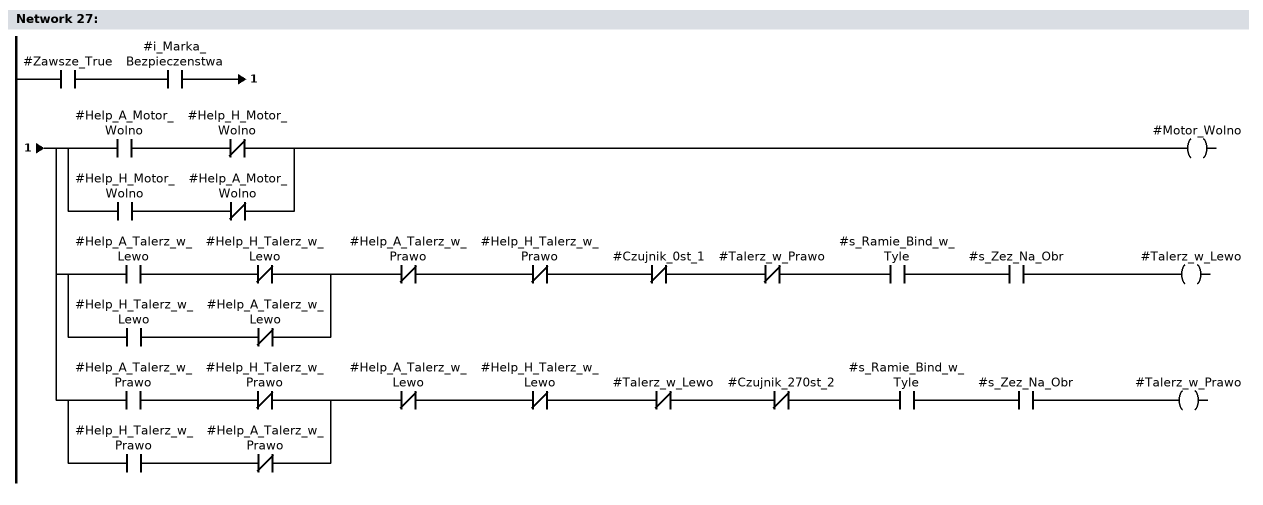
[picture p506: Obr_Na_Poz_4 networks 27-27]
NETWORK
TITLE =
//wykonianie obrotu warunki jazdy
      A     #Zawsze_True;
      A     #i_Marka_Bezpieczenstwa;
      =     L 1.0;
      A     L 1.0;
      A(;
      A     #Help_A_Motor_Wolno;
      AN    #Help_H_Motor_Wolno;
      O;
      A     #Help_H_Motor_Wolno;
      AN    #Help_A_Motor_Wolno;
      );
      =     #Motor_Wolno;
      A     L 1.0;
      A(;
      A     #Help_A_Talerz_w_Lewo;
      AN    #Help_H_Talerz_w_Lewo;
      O;
      A     #Help_H_Talerz_w_Lewo;
      AN    #Help_A_Talerz_w_Lewo;
      );
      AN    #Help_A_Talerz_w_Prawo;
      AN    #Help_H_Talerz_w_Prawo;
      AN    #Czujnik_0st_1;
      AN    #Talerz_w_Prawo;
      A     #s_Ramie_Bind_w_Tyle;
      A     #s_Zez_Na_Obr;
      =     #Talerz_w_Lewo;
      A     L 1.0;
      A(;
      A     #Help_A_Talerz_w_Prawo;
      AN    #Help_H_Talerz_w_Prawo;
      O;
      A     #Help_H_Talerz_w_Prawo;
      AN    #Help_A_Talerz_w_Prawo;
      );
      AN    #Help_A_Talerz_w_Lewo;
      AN    #Help_H_Talerz_w_Lewo;
      AN    #Talerz_w_Lewo;
      AN    #Czujnik_270st_2;
      A     #s_Ramie_Bind_w_Tyle;
      A     #s_Zez_Na_Obr;
      =     #Talerz_w_Prawo;
END_FUNCTION_BLOCK

FUNCTION_BLOCK "Pozycjonowanie_Bandy"	// FB 55
//Funcja odpowiada za jazde rolek na pozycje zgodnie z rozkazem 
VERSION : 0.1
VAR_INPUT
  i_Auto_Reczny : BOOL ;
  Stop_Bezpieczenistwa : BOOL ;
  Pozycjonuj_Lewo : BOOL ;
  Pozycjonuj_Prawo : BOOL ;
  Powrot_Poz : BOOL ;
  Foto_Przod : BOOL ;
  Foto_Tyl : BOOL ;
  i_Zez_Na_Rolki : BOOL ;
  Reset : BOOL ;
  Czas_Prawo : TIME ;
  Czas_Lewo : TIME ;
  Czas_Kontrolny : TIME ;
  Czas_Pow_Prawo : TIME ;
  Czas_Pow_Lewo : TIME ;
  Blokada_Obrotu_1 : BOOL ;
  i_Resetuj_Srodek : BOOL ;	//Przesow rolek z innego trybu
END_VAR
VAR_OUTPUT
  Potw_Pozycji : BOOL ;
  Pozycja_Lewo : BOOL ;	//Odniesienie do 0st
  Pozycja_Prawo : BOOL ;	//Odniesienie do 0st
  Pozycja_Srodek : BOOL ;
  Motor_Lewo : BOOL ;
  Motor_Prawo : BOOL ;
  Motor_Wolno : BOOL ;
  Zez_Na_Obrot : BOOL ;
  Blad_Pozycjowania : BOOL ;
END_VAR
VAR
  Pozycja_Wyjsciowa : BOOL ;
  Tim_Jazdy_Prawo : FB 20;
  Tim_Jazdy_Lewo : FB 20;
  Tim_Kon_Prawo : FB 20;	//Timmer kontrolny prawo
  Tim_Kon_Lewo : FB 20;	//Timmer kontrolny lewo
  Help_Motor_Prawo : BOOL ;
  Help_Motor_Lewo : BOOL ;
  H_Repozycj_Prawo : BOOL ;
  H_Repozycj_Lewo : BOOL ;
  Help_Motor_Wolno : BOOL ;
  H_Powr_od_Prawo_1 : BOOL ;
  H_Powr_od_Lewo_1 : BOOL ;
  H_Powr_Prawo : BOOL ;
  H_Powr_Lewo : BOOL ;
  Help_Poz_Prawo : BOOL ;
  Help_Poz_Lewo : BOOL ;
  Pozycj_Warunkowe : BOOL ;
  Skrajne_Prawo : BOOL ;
  Skrajne_Lewo : BOOL ;
  Zbocze_1 : BOOL ;
  Zbocze_2 : BOOL ;
  H6 : BOOL ;
  H7 : BOOL ;
  H8 : BOOL ;
  H9 : BOOL ;
  H10 : BOOL ;
END_VAR
VAR_TEMP
  Temp_Help_1 : BOOL ;
  Temp_Help_2 : BOOL ;
  Temp_Help_3 : BOOL ;
  Czas_Aktualny : TIME ;
END_VAR
BEGIN
NETWORK
TITLE =
      A     #Foto_Przod;
      A     #Foto_Tyl;
      A     #Pozycja_Srodek;
      A     #i_Zez_Na_Rolki;	//rolki sa odblokowane w pozycji 0st lub 180st
      =     #Pozycja_Wyjsciowa;
      O     #Help_Motor_Lewo;
      O     #Help_Motor_Prawo;
      R     #Potw_Pozycji;
//warunkowe pozycjonowanie 
NETWORK
TITLE =
//Pozycjonowanie prawo
//Pozycjonowanie w prawo
      A     #i_Zez_Na_Rolki;
      A     #Pozycjonuj_Prawo;
      A     #Pozycja_Wyjsciowa;
      S     #Help_Motor_Prawo;
      S     #Help_Motor_Wolno;
      S     #Help_Poz_Prawo;
      R     #Pozycja_Srodek;
      CALL  #Tim_Jazdy_Prawo (
           IN                       := #Help_Poz_Prawo,
           STOP                     := #Stop_Bezpieczenistwa,
           PT                       := #Czas_Prawo,
           Q_0                      := #Temp_Help_2,
           ET                       := #Czas_Aktualny);
      A     #Temp_Help_2;
      O;
      A     #Help_Poz_Prawo;
      AN    #Foto_Przod;
      S     #Pozycja_Prawo;
      S     #Potw_Pozycji;
      R     #Help_Motor_Prawo;
      R     #Help_Motor_Wolno;
      R     #Help_Poz_Prawo;
//Powrot z pozycjonowania. 
//Zjazd z fotokomorki aby zrobic ponowny najazd
      O(;
      A     #Foto_Przod;
      A     #Pozycja_Prawo;
      A     #Powrot_Poz;
      AN    #H_Powr_od_Prawo_1;
      );
      O(;
      A     #Pozycj_Warunkowe;
      );
      S     #Help_Motor_Prawo;
      S     #Help_Motor_Wolno;
      S     #H_Repozycj_Prawo;
      R     #Pozycja_Prawo;
//koniec zjazdu z fotokomorki
      AN    #Foto_Przod;
      A     #H_Repozycj_Prawo;
      R     #Help_Motor_Prawo;
      R     #Help_Motor_Wolno;
      R     #H_Repozycj_Prawo;
      S     #Skrajne_Prawo;
//powrot na pozycje na srodku obrtnicy
      A(;
      O     #Powrot_Poz;
      O     #Skrajne_Prawo;
      O     #Pozycj_Warunkowe;
      );
      A(;
      O     #Pozycja_Prawo;
      O     #Skrajne_Prawo;
      );
      AN    #Foto_Przod;
      S     #Help_Motor_Lewo;
      S     #Help_Motor_Wolno;
      S     #H_Powr_od_Prawo_1;
      R     #Help_Motor_Prawo;
      R     #Pozycja_Prawo;
      R     #Skrajne_Prawo;
      R     #Pozycj_Warunkowe;
NETWORK
TITLE =
//Pozycjonowanie lewo
//
//
//Pozycjonowanie w lewo
      A     #i_Zez_Na_Rolki;
      A     #Pozycjonuj_Lewo;
      A     #Pozycja_Wyjsciowa;
      S     #Help_Motor_Lewo;
      S     #Help_Motor_Wolno;
      S     #Help_Poz_Lewo;
      R     #Pozycja_Srodek;
      CALL  #Tim_Jazdy_Lewo (
           IN                       := #Help_Poz_Lewo,
           STOP                     := #Stop_Bezpieczenistwa,
           PT                       := #Czas_Lewo,
           Q_0                      := #Temp_Help_2,
           ET                       := #Czas_Aktualny);
      A     #Temp_Help_2;
      O;
      AN    #Foto_Tyl;
      A     #Help_Poz_Lewo;
      S     #Pozycja_Lewo;
      S     #Potw_Pozycji;
      R     #Help_Motor_Lewo;
      R     #Help_Motor_Wolno;
      R     #Help_Poz_Lewo;
//Powrot z pozycjonowania. 
//Zjazd z fotokomorki aby zrobic ponowny najazd
      A     #Foto_Tyl;
      A     #Pozycja_Lewo;
      A     #Powrot_Poz;
      AN    #H_Powr_od_Lewo_1;
      S     #Help_Motor_Lewo;
      S     #Help_Motor_Wolno;
      S     #H_Repozycj_Lewo;
      R     #Potw_Pozycji;
//koniec zjazdu z fotokomorki
      AN    #Foto_Tyl;
      A     #H_Repozycj_Lewo;
      R     #Help_Motor_Lewo;
      R     #Help_Motor_Wolno;
      R     #H_Repozycj_Lewo;
      S     #Skrajne_Lewo;
//powrot na pozycje na srodku obrotnicy
      O     #Skrajne_Lewo;
      O(;
      A     #Powrot_Poz;
      A     #Pozycja_Lewo;
      );
      AN    #Foto_Tyl;
      S     #Help_Motor_Prawo;
      S     #Help_Motor_Wolno;
      S     #H_Powr_od_Lewo_1;
      R     #Help_Motor_Lewo;
      R     #Pozycja_Lewo;
      R     #Skrajne_Lewo;
NETWORK
TITLE =
//Okreselnie srodka
//Jazda  powrotna w strone prawa do œrodka
      A     #Foto_Przod;
      A     #H_Powr_od_Prawo_1;
      S     #H_Powr_Prawo;
      CALL  #Tim_Kon_Prawo (
           IN                       := #H_Powr_Prawo,
           STOP                     := #Stop_Bezpieczenistwa,
           PT                       := #Czas_Pow_Prawo,
           Q_0                      := #Temp_Help_2,
           ET                       := #Czas_Aktualny);
      A     #Foto_Tyl;
      A     #H_Powr_od_Lewo_1;
      S     #H_Powr_Lewo;
      CALL  #Tim_Kon_Lewo (
           IN                       := #H_Powr_Lewo,
           STOP                     := #Stop_Bezpieczenistwa,
           PT                       := #Czas_Pow_Lewo,
           Q_0                      := #Temp_Help_3,
           ET                       := #Czas_Aktualny);
//nieautoryzowane kasowanie srodka
      A     #i_Resetuj_Srodek;
      FP    #Zbocze_2;
      R     #Pozycja_Srodek;
      O     #Temp_Help_3;
      O     #Temp_Help_2;
      S     #Pozycja_Srodek;
      S     #Potw_Pozycji;
      R     #Pozycj_Warunkowe;
//zresetuj bity i pozycjonuj do srodka
      A     #Reset;
      FP    #Zbocze_1;
      S     #Pozycj_Warunkowe;
      R     #Pozycja_Srodek;
      R     #Potw_Pozycji;
      =     #Temp_Help_1;
      O     #Temp_Help_1;
      O     #Temp_Help_2;
      O     #Temp_Help_3;
      R     #Help_Motor_Prawo;
      R     #Help_Motor_Lewo;
      R     #Help_Motor_Wolno;
      R     #H_Powr_od_Prawo_1;
      R     #H_Powr_od_Lewo_1;
      R     #H_Repozycj_Prawo;
      R     #H_Repozycj_Lewo;
      R     #Help_Poz_Prawo;
      R     #Help_Poz_Lewo;
      R     #Skrajne_Prawo;
      R     #Skrajne_Lewo;
      R     #H_Powr_Prawo;
      R     #H_Powr_Lewo;
      R     #Pozycja_Prawo;
      R     #Pozycja_Lewo;
NETWORK
TITLE =
//Przyporzadkowanie wyjsc
      A     #i_Auto_Reczny;
      A     #i_Zez_Na_Rolki;
      A     #Help_Motor_Lewo;
      =     #Motor_Lewo;
      A     #i_Auto_Reczny;
      A     #i_Zez_Na_Rolki;
      A     #Help_Motor_Prawo;
      =     #Motor_Prawo;
      A     #i_Auto_Reczny;
      A     #Help_Motor_Wolno;
      =     #Motor_Wolno;
//Zezwolenie na obrot obrotnicy
      A(;
      A     #Foto_Przod;
      A     #Foto_Tyl;
      O;
      AN    #Foto_Przod;
      AN    #Foto_Tyl;
      );
      A     #Blokada_Obrotu_1;
      =     #Zez_Na_Obrot;
END_FUNCTION_BLOCK

FUNCTION_BLOCK "Bindownica_Test"	// FB 57
VERSION : 0.1
VAR_INPUT
  i_Bind_Obwod_Ok : BOOL ;	//270 stopni
  i_Bind_Poz_Podst : BOOL ;
  i_Bind_Syg_Got : BOOL ;
  i_Bind_Blad : BOOL ;
  i_Bind_Start_Kon : BOOL ;	//Bindownica start koniec wiazania
  i_Przesznuruj : BOOL ;	//Przesznurowanie imituje bindownice
  i_Cykl_Bindowanie : BOOL ;
END_VAR
VAR_OUTPUT
  io_Bind_Obwod_Ok : BOOL ;	//270 stopni
  io_Bind_Poz_Podst : BOOL ;
  io_Bind_Syg_Got : BOOL ;
  io_Bind_Blad : BOOL ;
  io_Bind_Start_Kon : BOOL ;	//Bindownica start koniec wiazania
END_VAR
VAR
  CZas_Testowy : SFB 4;
END_VAR
VAR_TEMP
  temp_help_1 : BOOL ;
END_VAR
BEGIN
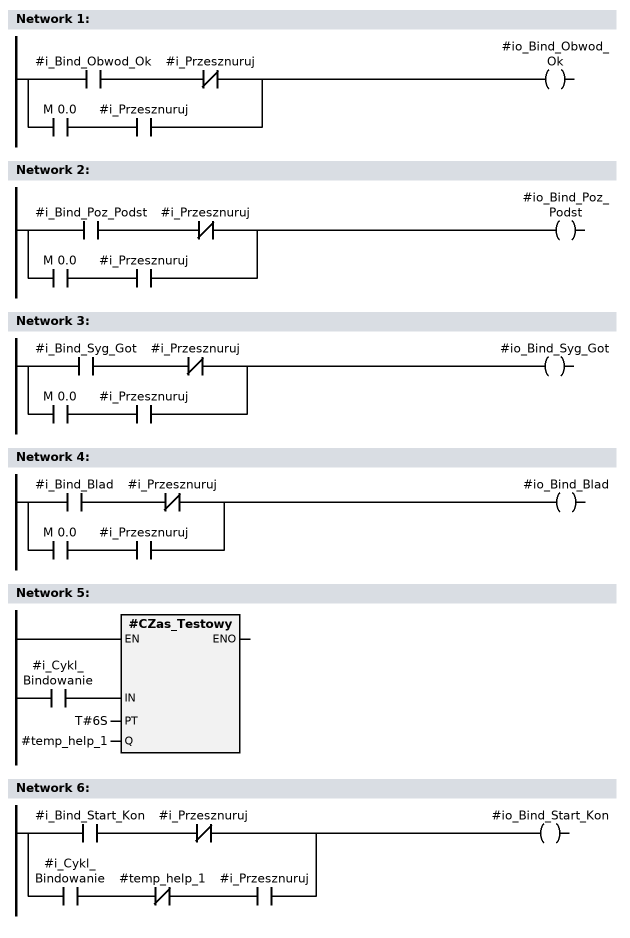
NETWORK
TITLE =
//bind obwod ok
      A     #i_Bind_Obwod_Ok;
      AN    #i_Przesznuruj;
      O;
      A     M 0.0;
      A     #i_Przesznuruj;
      =     #io_Bind_Obwod_Ok;
NETWORK
TITLE =
//Pozycja podstawowa
      A     #i_Bind_Poz_Podst;
      AN    #i_Przesznuruj;
      O;
      A     M 0.0;
      A     #i_Przesznuruj;
      =     #io_Bind_Poz_Podst;
NETWORK
TITLE =
//sygnal gotowosc
      A     #i_Bind_Syg_Got;
      AN    #i_Przesznuruj;
      O;
      A     M 0.0;
      A     #i_Przesznuruj;
      =     #io_Bind_Syg_Got;
NETWORK
TITLE =
//Blad bindowania
      A     #i_Bind_Blad;
      AN    #i_Przesznuruj;
      O;
      A     M 0.0;
      A     #i_Przesznuruj;
      =     #io_Bind_Blad;
NETWORK
TITLE =
//bindowanie
//
      A     #i_Cykl_Bindowanie;
      =     L 1.0;
      BLD   103;
      CALL  #CZas_Testowy (
           IN                       := L 1.0,
           PT                       := T#6S,
           Q                        := #temp_help_1);
      NOP   0;
NETWORK
TITLE =
//start koniec bindowania
      A     #i_Bind_Start_Kon;
      AN    #i_Przesznuruj;
      O;
      A     #i_Cykl_Bindowanie;
      AN    #temp_help_1;
      A     #i_Przesznuruj;
      =     #io_Bind_Start_Kon;
END_FUNCTION_BLOCK

FUNCTION_BLOCK "Pozycjonowanie_Palety"	// FB 58
//Funcja odpowiada za jazde rolek na pozycje zgodnie z rozkazem. Zmiany do wersji 
//porzednie:
//
//-o powrocie z pozycjonowania gdy stan pozycji palety jest nieustalony decyduje
// bit wejsciowy reset
//
VERSION : 0.1
VAR_INPUT
  i_Marka_Bezpieczenstwa : BOOL ;
  i_Rezerwa : BOOL ;
  i_Auto_Reczny : BOOL ;
  i_Pozycjonuj_Lewo : BOOL ;
  i_Pozycjonuj_Prawo : BOOL ;
  i_Pozycjonuj_Srodek : BOOL ;
  i_Foto_Przod : BOOL ;
  i_Foto_Tyl : BOOL ;
  s_i_Zez_Na_Rolki : BOOL ;
  i_Czas_Jazdy_Prawo : TIME ;
  i_Czas_Jazdy_Lewo : TIME ;
  i_Czas_Opoznienia : TIME ;
  i_Czas_Powrotu_Prawo : TIME ;
  i_Czas_Powrotu_Lewo : TIME ;
  s_i_Blokada_Obrotu : BOOL ;
  i_Resetuj_Srodek : BOOL ;	//Resetowanie zewnetrzne konca palety
  i_Setuj_Srodek : BOOL ;	//Ustawienie zewnetrzne srodka palety
END_VAR
VAR_OUTPUT
  o_Pozycja_Lewo : BOOL ;	//Odniesienie do 0st
  o_Pozycja_Prawo : BOOL ;	//Odniesienie do 0st
  o_Pozycja_Srodek : BOOL ;
  o_Potw_Pozycji : BOOL ;
  o_Motor_Lewo : BOOL ;
  o_Motor_Prawo : BOOL ;
  o_Motor_Wolno : BOOL ;
  s_o_Zez_Na_Obrot : BOOL ;
  o_Rezerwa_1 : BOOL ;
  o_Rezerwa_2 : BOOL ;
  o_Rezerwa_3 : BOOL ;
END_VAR
VAR
  Tim_Jazdy_Lewo : FB 20;
  Tim_Jazdy_Prawo : FB 20;
  Tim_Kon_Prawo : FB 20;	//Timmer kontrolny prawo
  Tim_Kon_Lewo : FB 20;	//Timmer kontrolny lewo
  Tim_Opoznienia : FB 20;
  Stop_Czas_Kontrolny : BOOL ;
  Help_Motor_Prawo : BOOL ;
  Help_Motor_Lewo : BOOL ;
  Help_Motor_Wolno : BOOL ;
  H_Repozycj_Prawo : BOOL ;
  H_Repozycj_Lewo : BOOL ;
  H_Powrot_od_Prawej : BOOL ;
  H_Powrot_od_Lewej : BOOL ;
  H_Czas_Powr_Prawo : BOOL ;
  H_Czas_Powr_Lewo : BOOL ;
  H_Czas_Jazdy_Prawo : BOOL ;
  H_Czas_Jazdy_Lewo : BOOL ;
  H_Krawedz_Prawo : BOOL ;
  H_Krawedz_Lewo : BOOL ;
  H_Pozycja_Wyjsciowa : BOOL ;
  H_Brak_Pozycji : BOOL ;
  Zbocze_1 : BOOL ;
  Zbocze_2 : BOOL ;
  H_Jakas_Pozycja : BOOL ;
  H8 : BOOL ;
  H9 : BOOL ;
  H10 : BOOL ;
  H11 : BOOL ;
  H12 : BOOL ;
END_VAR
VAR_TEMP
  Temp_Help_1 : BOOL ;
  Temp_Help_2 : BOOL ;
  Temp_Help_3 : BOOL ;
  Temp_Help_4 : BOOL ;
  Czas_Aktualny : TIME ;
END_VAR
BEGIN
NETWORK
TITLE =
//Ten network celowo ma byc wolny
NETWORK
TITLE =
//Zatrzymanie czasu w timmerach gdy obwod bezpieczenstwa nie ok
      A     #i_Marka_Bezpieczenstwa;
      S     #Stop_Czas_Kontrolny;
      AN    #i_Marka_Bezpieczenstwa;
      AN    #Stop_Czas_Kontrolny;
      JC    end;
      AN    #i_Marka_Bezpieczenstwa;
      R     #Stop_Czas_Kontrolny;
NETWORK
TITLE =
      A     #i_Foto_Przod;
      A     #i_Foto_Tyl;
      A     #o_Pozycja_Srodek;
      A     #s_i_Zez_Na_Rolki;	//rolki sa odblokowane w pozycji 0st lub 180st
      =     #H_Pozycja_Wyjsciowa;
//Reset pozycji gdy silnki wykonaja ruch
      O     #Help_Motor_Lewo;
      O     #Help_Motor_Prawo;
      R     #o_Pozycja_Prawo;
      R     #o_Pozycja_Srodek;
      R     #o_Pozycja_Lewo;
//warunkowe pozycjonowanie brak pozycji
      AN    #o_Pozycja_Prawo;
      AN    #o_Pozycja_Lewo;
      AN    #o_Pozycja_Srodek;
      =     #H_Brak_Pozycji;
      NOT;
      =     #H_Jakas_Pozycja;
NETWORK
TITLE =
//Pozycjonowanie prawo
//Pozycjonowanie w prawo
      A     #i_Pozycjonuj_Prawo;
      AN    #i_Pozycjonuj_Srodek;
      AN    #i_Pozycjonuj_Lewo;
      A     #H_Pozycja_Wyjsciowa;
      S     #Help_Motor_Prawo;
      R     #Help_Motor_Lewo;
      S     #H_Czas_Jazdy_Prawo;
//Uruchom zjazd z fotokomorki
      CALL  #Tim_Jazdy_Prawo (
           IN                       := #H_Czas_Jazdy_Prawo,
           STOP                     := #Stop_Czas_Kontrolny,
           PT                       := #i_Czas_Jazdy_Prawo,
           Q_0                      := #Temp_Help_2,
           ET                       := #Czas_Aktualny);
      A     #Temp_Help_2;
      O;
      A     #H_Czas_Jazdy_Prawo;
      AN    #i_Foto_Przod;
      S     #o_Pozycja_Prawo;
      R     #Help_Motor_Prawo;
      R     #H_Czas_Jazdy_Prawo;
NETWORK
TITLE =
//Powrot ze strony prawej
//Powrot z pozycjonowania. 
//Zjazd z fotokomorki aby zrobic ponowny najazd
      O     #o_Pozycja_Prawo;
      O     #H_Brak_Pozycji;
      A     #i_Pozycjonuj_Srodek;
      A     #i_Foto_Przod;
      A     #i_Foto_Tyl;
      A     #s_i_Zez_Na_Rolki;
      AN    #H_Powrot_od_Prawej;
      S     #Help_Motor_Prawo;
      S     #H_Repozycj_Prawo;
      R     #Help_Motor_Lewo;
//koniec zjazdu z fotokomorki
      AN    #i_Foto_Przod;
//      A     #H_Repozycj_Prawo
      R     #Help_Motor_Prawo;
      R     #H_Repozycj_Prawo;
      S     #H_Krawedz_Prawo;
//powrot na pozycje na srodku obrotnicy
      A(;
      O     #i_Pozycjonuj_Srodek;
      O     #H_Krawedz_Prawo;
      );
      A(;
      O     #o_Pozycja_Prawo;
      O     #H_Krawedz_Prawo;
      );
      AN    #i_Foto_Przod;
      S     #Help_Motor_Lewo;
      S     #H_Powrot_od_Prawej;
      R     #Help_Motor_Prawo;
      R     #H_Krawedz_Prawo;
NETWORK
TITLE =
//Pozycjonowanie lewo
//
//
//Pozycjonowanie w lewo
      A     #i_Pozycjonuj_Lewo;
      AN    #i_Pozycjonuj_Srodek;
      AN    #i_Pozycjonuj_Prawo;
      A     #H_Pozycja_Wyjsciowa;
      S     #Help_Motor_Lewo;
      R     #Help_Motor_Prawo;
      S     #H_Czas_Jazdy_Lewo;
      CALL  #Tim_Jazdy_Lewo (
           IN                       := #H_Czas_Jazdy_Lewo,
           STOP                     := #Stop_Czas_Kontrolny,
           PT                       := #i_Czas_Jazdy_Lewo,
           Q_0                      := #Temp_Help_2,
           ET                       := #Czas_Aktualny);
      A     #Temp_Help_2;
      O;
      A     #H_Czas_Jazdy_Lewo;
      AN    #i_Foto_Tyl;
      S     #o_Pozycja_Lewo;
      R     #Help_Motor_Lewo;
      R     #H_Czas_Jazdy_Lewo;
NETWORK
TITLE =
//Powrot ze strony lewej
//Powrot z pozycjonowania. 
//Zjazd z fotokomorki aby zrobic ponowny najazd
      A     #i_Pozycjonuj_Srodek;
      A     #i_Foto_Przod;
      A     #i_Foto_Tyl;
      A     #o_Pozycja_Lewo;
      A     #s_i_Zez_Na_Rolki;
      AN    #H_Powrot_od_Lewej;
      S     #Help_Motor_Lewo;
      R     #Help_Motor_Prawo;
      S     #H_Repozycj_Lewo;
//koniec zjazdu z fotokomorki
      AN    #i_Foto_Tyl;
      A     #H_Repozycj_Lewo;
      R     #Help_Motor_Lewo;
      R     #H_Repozycj_Lewo;
      S     #H_Krawedz_Lewo;
//powrot na pozycje na srodku obrotnicy
      O     #H_Krawedz_Lewo;
      O(;
      A     #i_Pozycjonuj_Srodek;
      A     #o_Pozycja_Lewo;
      );
      AN    #i_Foto_Tyl;
      S     #Help_Motor_Prawo;
      S     #H_Powrot_od_Lewej;
      R     #Help_Motor_Lewo;
      R     #H_Krawedz_Lewo;
NETWORK
TITLE =
//Okreselnie srodka
//Jazda  powrotna w strone prawa do œrodka
      A     #i_Foto_Przod;
      A     #H_Powrot_od_Prawej;
      S     #H_Czas_Powr_Prawo;
      CALL  #Tim_Kon_Prawo (
           IN                       := #H_Czas_Powr_Prawo,
           STOP                     := #Stop_Czas_Kontrolny,
           PT                       := #i_Czas_Powrotu_Prawo,
           Q_0                      := #Temp_Help_1,
           ET                       := #Czas_Aktualny);
//Powrot ze strony lewej do srodka
      A     #i_Foto_Tyl;
      A     #H_Powrot_od_Lewej;
      S     #H_Czas_Powr_Lewo;
      CALL  #Tim_Kon_Lewo (
           IN                       := #H_Czas_Powr_Lewo,
           STOP                     := #Stop_Czas_Kontrolny,
           PT                       := #i_Czas_Powrotu_Lewo,
           Q_0                      := #Temp_Help_2,
           ET                       := #Czas_Aktualny);
//nieautoryzowane kasowanie srodka
      A     #i_Resetuj_Srodek;
      R     #o_Pozycja_Srodek;
      =     #Temp_Help_3;
//nieautoryzowane setowanie  srodka
      A     #i_Setuj_Srodek;
      FP    #Zbocze_1;
      A     #i_Foto_Przod;
      A     #i_Foto_Tyl;
      S     #o_Pozycja_Srodek;
      =     #Temp_Help_4;
      O     #Temp_Help_1;
      O     #Temp_Help_2;
      S     #o_Pozycja_Srodek;
//Reset wszystkich zbedncyh bitow
      O     #Temp_Help_1;
      O     #Temp_Help_2;
      O     #Temp_Help_3;
      O     #Temp_Help_4;
      R     #Help_Motor_Prawo;
      R     #Help_Motor_Lewo;
      R     #H_Powrot_od_Prawej;
      R     #H_Powrot_od_Lewej;
      R     #H_Repozycj_Prawo;
      R     #H_Repozycj_Lewo;
      R     #H_Czas_Jazdy_Prawo;
      R     #H_Czas_Jazdy_Lewo;
      R     #H_Krawedz_Prawo;
      R     #H_Krawedz_Lewo;
      R     #H_Czas_Powr_Prawo;
      R     #H_Czas_Powr_Lewo;
      R     #o_Pozycja_Prawo;
      R     #o_Pozycja_Lewo;
NETWORK
TITLE =
//Jezeli dluzej niz 1.5 sekundy to pozycja potwierdzona
      CALL  #Tim_Opoznienia (
           IN                       := #H_Jakas_Pozycja,
           STOP                     := #Stop_Czas_Kontrolny,
           PT                       := T#1S500MS,
           Q_0                      := #o_Potw_Pozycji);
NETWORK
TITLE =
//Przyporzadkowanie wyjsc
end:  NOP   0;
//-
      A     #i_Auto_Reczny;
      A     #i_Marka_Bezpieczenstwa;
      A     #s_i_Zez_Na_Rolki;
      A     #Help_Motor_Lewo;
      AN    #Help_Motor_Prawo;
      =     #o_Motor_Lewo;
//-
      A     #i_Auto_Reczny;
      A     #i_Marka_Bezpieczenstwa;
      A     #s_i_Zez_Na_Rolki;
      A     #Help_Motor_Prawo;
      AN    #Help_Motor_Lewo;
      =     #o_Motor_Prawo;
//-
      O     #o_Motor_Lewo;
      O     #o_Motor_Prawo;
      =     #o_Motor_Wolno;
//Zezwolenie na obrot obrotnicy
      A(;
      A     #i_Foto_Przod;
      A     #i_Foto_Tyl;
      O;
      AN    #i_Foto_Przod;
      AN    #i_Foto_Tyl;
      );
      A     #s_i_Blokada_Obrotu;
      =     #s_o_Zez_Na_Obrot;
END_FUNCTION_BLOCK

FUNCTION "Funkcja_Bezpieczenstwa" : VOID	// FC 3
//Funkcja steruje bezpieczenstwem maszyny
VERSION : 0.1
VAR_TEMP
  Help_Bit : BOOL ;
END_VAR
BEGIN
NETWORK
TITLE =
//Ten Network celowo jest wolny
//
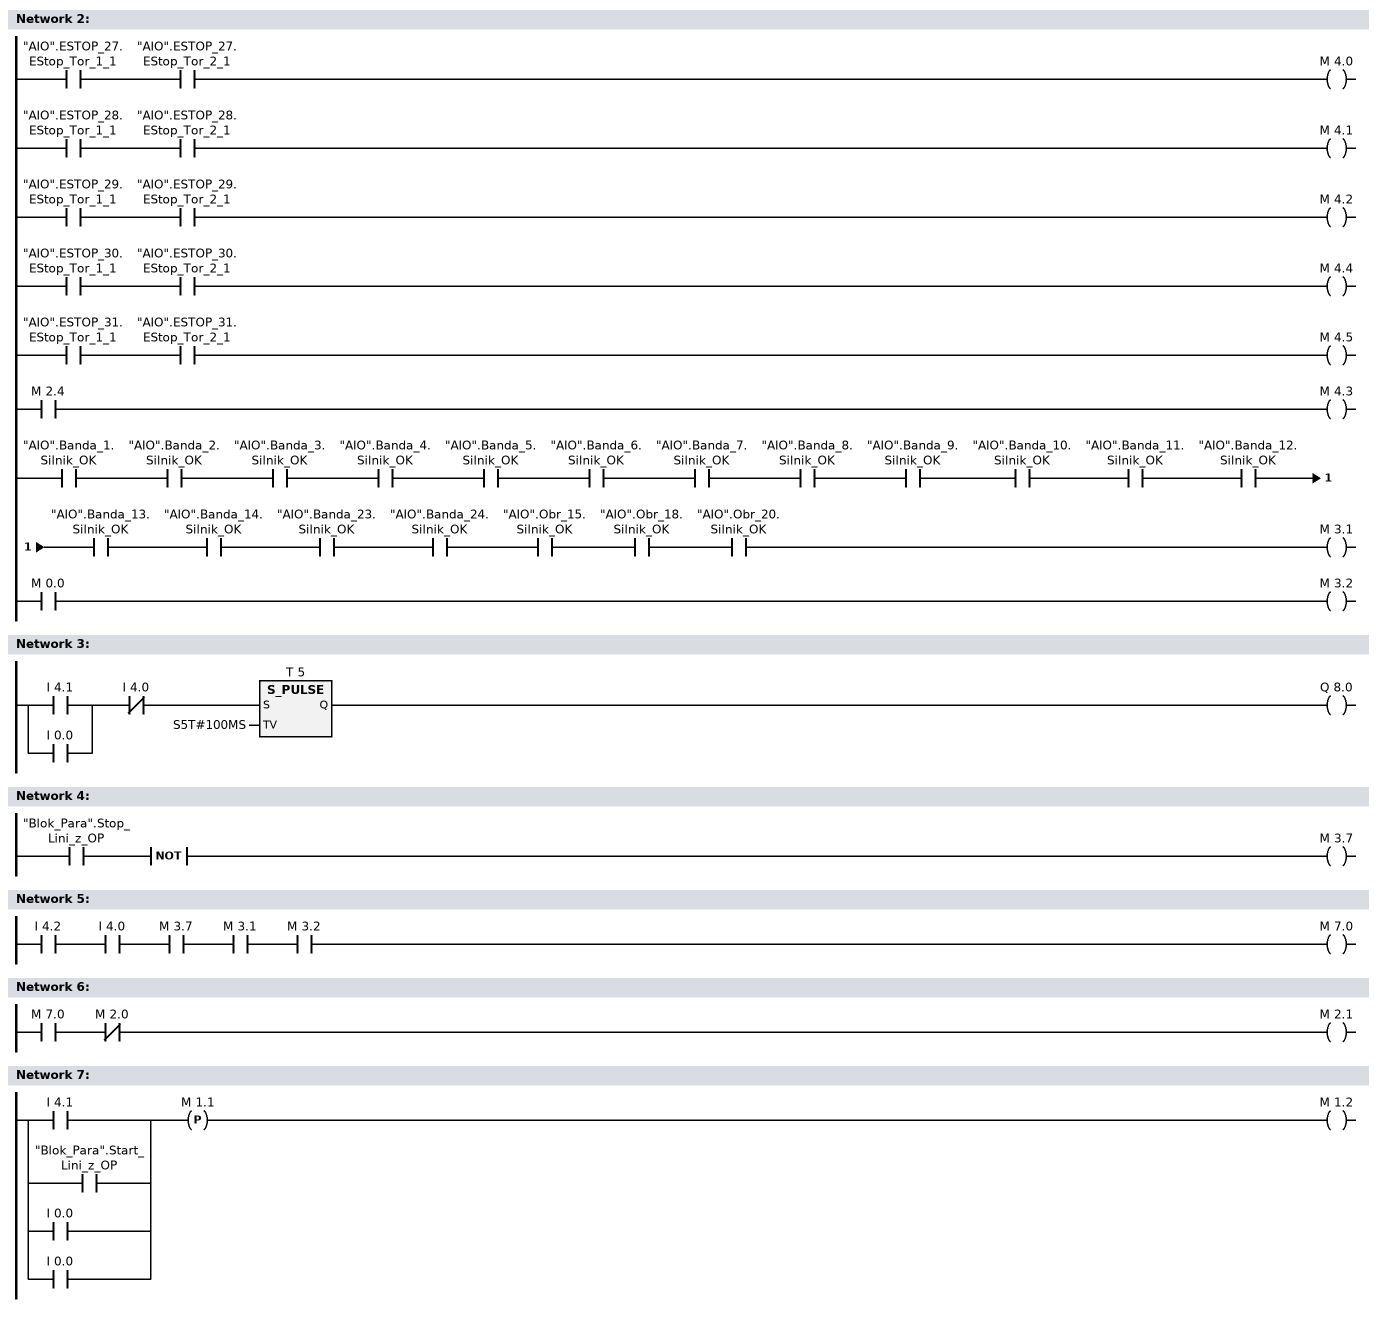
NETWORK
TITLE =
//Not Aus 27*******************************
      A     "AIO".ESTOP_27.EStop_Tor_1_1;
      A     "AIO".ESTOP_27.EStop_Tor_2_1;
      =     M 4.0;
//Not Aus 28*******************************
      A     "AIO".ESTOP_28.EStop_Tor_1_1;
      A     "AIO".ESTOP_28.EStop_Tor_2_1;
      =     M 4.1;
//Not Aus 29*******************************
      A     "AIO".ESTOP_29.EStop_Tor_1_1;
      A     "AIO".ESTOP_29.EStop_Tor_2_1;
      =     M 4.2;
//Not Aus 30*******************************
      A     "AIO".ESTOP_30.EStop_Tor_1_1;
      A     "AIO".ESTOP_30.EStop_Tor_2_1;
      =     M 4.4;
//Not Aus 31*******************************
      A     "AIO".ESTOP_31.EStop_Tor_1_1;
      A     "AIO".ESTOP_31.EStop_Tor_2_1;
      =     M 4.5;
//Strefa *******************************
      A     M 2.4;
      =     M 4.3;
//Falowniki********************************
      A     "AIO".Banda_1.Silnik_OK;
      A     "AIO".Banda_2.Silnik_OK;
      A     "AIO".Banda_3.Silnik_OK;
      A     "AIO".Banda_4.Silnik_OK;
      A     "AIO".Banda_5.Silnik_OK;
      A     "AIO".Banda_6.Silnik_OK;
      A     "AIO".Banda_7.Silnik_OK;
      A     "AIO".Banda_8.Silnik_OK;
      A     "AIO".Banda_9.Silnik_OK;
      A     "AIO".Banda_10.Silnik_OK;
      A     "AIO".Banda_11.Silnik_OK;
      A     "AIO".Banda_12.Silnik_OK;
      A     "AIO".Banda_13.Silnik_OK;
      A     "AIO".Banda_14.Silnik_OK;
      A     "AIO".Banda_23.Silnik_OK;
      A     "AIO".Banda_24.Silnik_OK;
      A     "AIO".Obr_15.Silnik_OK;
      A     "AIO".Obr_18.Silnik_OK;
      A     "AIO".Obr_20.Silnik_OK;
      =     M 3.1;
//Bezpieczniki Szafa************************
//Brak w szafie bepiecznikow z kontrola wiec
      A     M 0.0;
      =     M 3.2;
NETWORK
TITLE =
//Reset przekaznika bezp
      A(;
      O     I 4.1;
      O     I 0.0;
      );
      AN    I 4.0;
      L     S5T#100MS;
      SP    T 5;
      NOP   0;
      NOP   0;
      NOP   0;
      A     T 5;
      =     Q 8.0;
NETWORK
TITLE =
      A     "Blok_Para".Stop_Lini_z_OP;
      NOT;
      =     M 3.7;
NETWORK
TITLE =
//Warunki Startu 
      A     I 4.2;
      A     I 4.0;
      A     M 3.7;
      A     M 3.1;
      A     M 3.2;
      =     M 7.0;
NETWORK
TITLE =
//warunki do strartu ok ale start nie wcisniety
      A     M 7.0;
      AN    M 2.0;
      =     M 2.1;
NETWORK
TITLE =
//Start na szafie glownej
      A(;
      O     I 4.1;
      O     "Blok_Para".Start_Lini_z_OP;
      O     I 0.0;
      O     I 0.0;
      );
      FP    M 1.1;
      =     M 1.2;
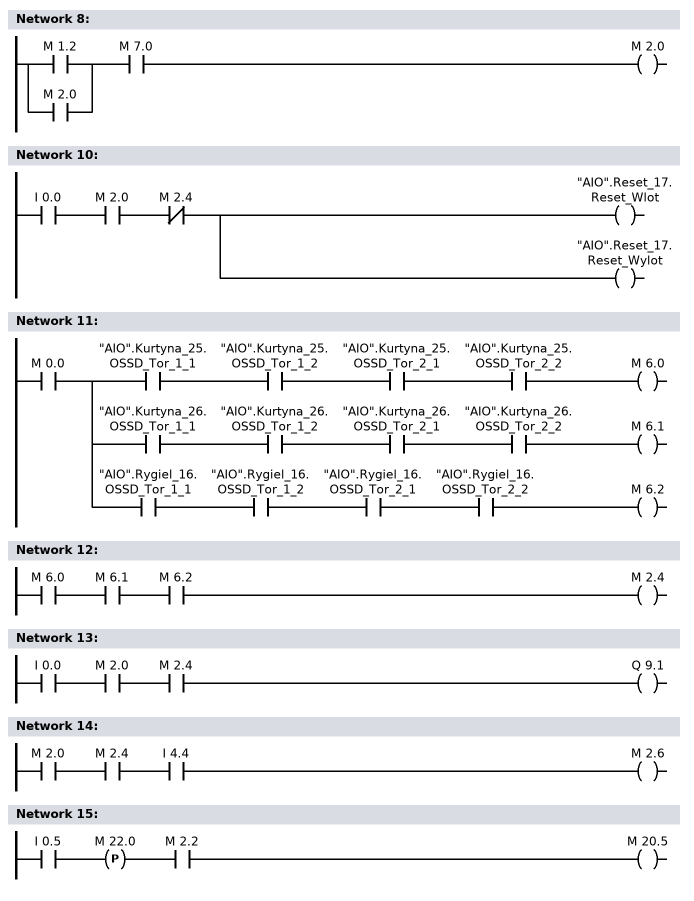
NETWORK
TITLE =
//Start Lini. Zalaczenie marki bezpieczenstwa
      A(;
      O     M 1.2;
      O     M 2.0;
      );
      A     M 7.0;
      =     M 2.0;
NETWORK
TITLE =
//Poczatek drugiego przekaznika bezpieczenstwa
NETWORK
TITLE =
//Resetowanie kurtyn bezpieczenstwa
//
      A     I 0.0;
      A     M 2.0;
      AN    M 2.4;
      =     "AIO".Reset_17.Reset_Wlot;
      =     "AIO".Reset_17.Reset_Wylot;
NETWORK
TITLE =
//Kurtyny wlot ok modul 25
//Kurtyny wylot ok modull 26
//Rygiel adres 16 ok
      A     M 0.0;
      =     L 1.0;
      A     L 1.0;
      A     "AIO".Kurtyna_25.OSSD_Tor_1_1;
      A     "AIO".Kurtyna_25.OSSD_Tor_1_2;
      A     "AIO".Kurtyna_25.OSSD_Tor_2_1;
      A     "AIO".Kurtyna_25.OSSD_Tor_2_2;
      =     M 6.0;
      A     L 1.0;
      A     "AIO".Kurtyna_26.OSSD_Tor_1_1;
      A     "AIO".Kurtyna_26.OSSD_Tor_1_2;
      A     "AIO".Kurtyna_26.OSSD_Tor_2_1;
      A     "AIO".Kurtyna_26.OSSD_Tor_2_2;
      =     M 6.1;
      A     L 1.0;
      A     "AIO".Rygiel_16.OSSD_Tor_1_1;
      A     "AIO".Rygiel_16.OSSD_Tor_1_2;
      A     "AIO".Rygiel_16.OSSD_Tor_2_1;
      A     "AIO".Rygiel_16.OSSD_Tor_2_2;
      =     M 6.2;
NETWORK
TITLE =
//Sprawdzenei czy strefa maszyny bindujacej bezpieczna
      A     M 6.0;
      A     M 6.1;
      A     M 6.2;
      =     M 2.4;
NETWORK
TITLE =
//Reset strefy bezpieczenstwa
      A     I 0.0;
      A     M 2.0;
      A     M 2.4;
      =     Q 9.1;
NETWORK
TITLE =
//Marka do pracy dla lini bindujacej
//Uwzglednione sa warunki kurtyn
//
      A     M 2.0;
      A     M 2.4;
      A     I 4.4;
      =     M 2.6;
NETWORK
TITLE =
//Tak aby potwierdzic stop gdy paleta na obrotnicy
      A     I 0.5;
      FP    M 22.0;
      A     M 2.2;
      =     M 20.5;
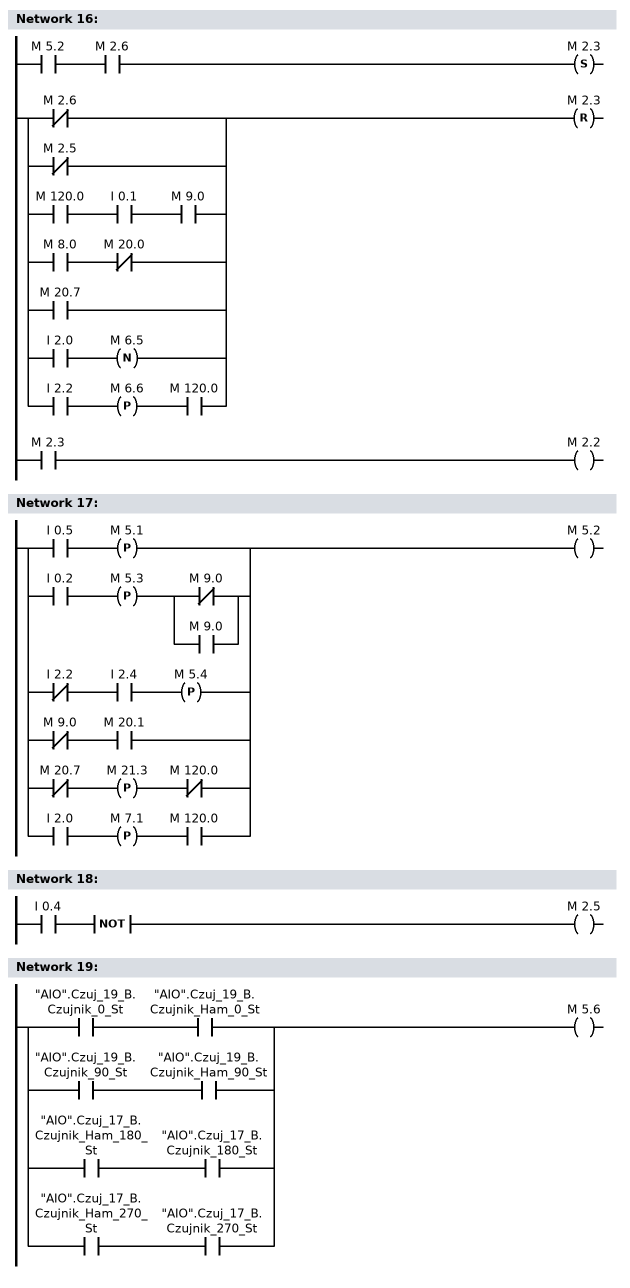
NETWORK
TITLE =
      A     M 5.2;
      A     M 2.6;
      S     M 2.3;
      A(;
      ON    M 2.6;
      ON    M 2.5;
      O(;
      A     M 120.0;
      A     I 0.1;
      A     M 9.0;
      );
      O(;
      A     M 8.0;
      AN    M 20.0;
      );
      O     M 20.7;
      O(;
      A     I 2.0;
      FN    M 6.5;
      );
      O(;
      A     I 2.2;
      FP    M 6.6;
      A     M 120.0;
      );
      );
      R     M 2.3;
      A     M 2.3;
      =     M 2.2;
NETWORK
TITLE =
//Cykl bindownicy przywrocenie
//Jest wiele drog do tego samego celu 
      A     I 0.5;
      FP    M 5.1;
      O(;
      A     I 0.2;
      FP    M 5.3;
      A(;
      ON    M 9.0;
      O     M 9.0;
      );
      );
      O(;
      AN    I 2.2;
      A     I 2.4;
      FP    M 5.4;
      );
      O(;
      AN    M 9.0;
      A     M 20.1;
      );
      O(;
      AN    M 20.7;
      FP    M 21.3;
      AN    M 120.0;
      );
      O(;
      A     I 2.0;
      FP    M 7.1;
      A     M 120.0;
      );
      =     M 5.2;
NETWORK
TITLE =
//Przycisk stop w automacie zatrzymuje maszyne 
      A     I 0.4;
      NOT;
      =     M 2.5;
NETWORK
TITLE =
//Wysuniecie OK
      A     "AIO".Czuj_19_B.Czujnik_0_St;
      A     "AIO".Czuj_19_B.Czujnik_Ham_0_St;
      O;
      A     "AIO".Czuj_19_B.Czujnik_90_St;
      A     "AIO".Czuj_19_B.Czujnik_Ham_90_St;
      O;
      A     "AIO".Czuj_17_B.Czujnik_Ham_180_St;
      A     "AIO".Czuj_17_B.Czujnik_180_St;
      O;
      A     "AIO".Czuj_17_B.Czujnik_Ham_270_St;
      A     "AIO".Czuj_17_B.Czujnik_270_St;
      =     M 5.6;
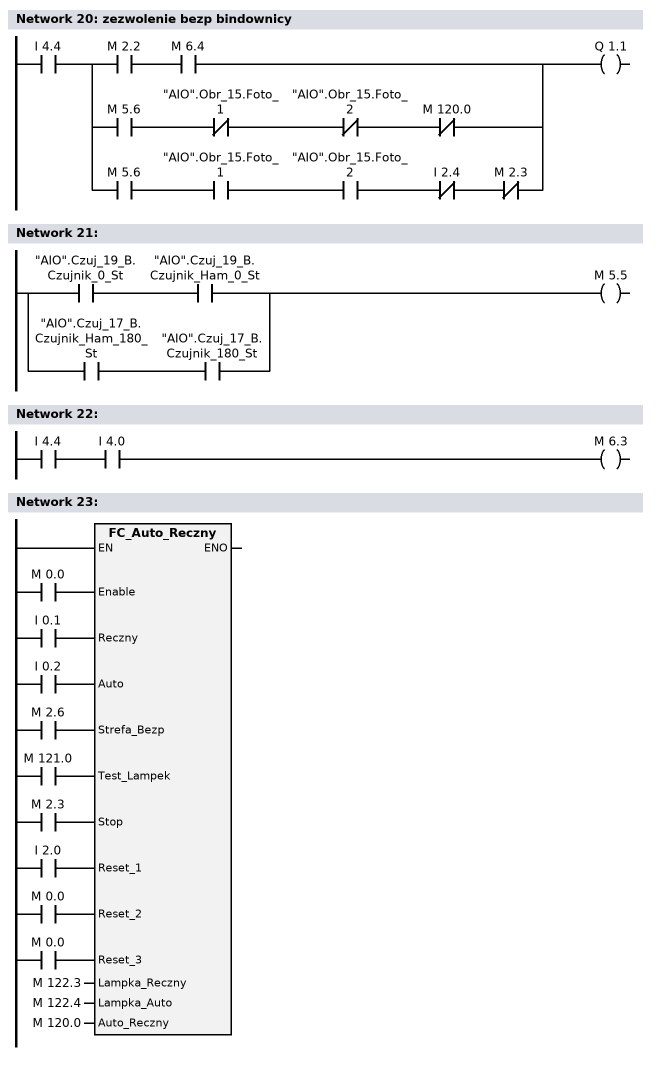
NETWORK
TITLE = zezwolenie bezp bindownicy
//Obwod bezpieczenstwa do bindownicy.
      A     I 4.4;
      A(;
      A     M 2.2;
      A     M 6.4;
      O;
      A     M 5.6;
      AN    "AIO".Obr_15.Foto_1;
      AN    "AIO".Obr_15.Foto_2;
      AN    M 120.0;
      O;
      A     M 5.6;
      A     "AIO".Obr_15.Foto_1;
      A     "AIO".Obr_15.Foto_2;
      AN    I 2.4;
      AN    M 2.3;
      );
      =     Q 1.1;
NETWORK
TITLE =
//Kat jazdy rolek ok 
      A     "AIO".Czuj_19_B.Czujnik_0_St;
      A     "AIO".Czuj_19_B.Czujnik_Ham_0_St;
      O;
      A     "AIO".Czuj_17_B.Czujnik_Ham_180_St;
      A     "AIO".Czuj_17_B.Czujnik_180_St;
      =     M 5.5;
NETWORK
TITLE =
//Sygnal imitujacy kurtyne i grzyba 
      A     I 4.4;
      A     I 4.0;
      =     M 6.3;
NETWORK
TITLE =
//Wybranie trybu pracy bindownicy (reczny/auto)
//Jezeli cos nie tak ze strefa to przejscie na reczny
      A     M 0.0;
      =     L 1.0;
      BLD   103;
      A     I 0.1;
      =     L 1.1;
      BLD   103;
      A     I 0.2;
      =     L 1.2;
      BLD   103;
      A     M 2.6;
      =     L 1.3;
      BLD   103;
      A     M 121.0;
      =     L 1.4;
      BLD   103;
      A     M 2.3;
      =     L 1.5;
      BLD   103;
      A     I 2.0;
      =     L 1.6;
      BLD   103;
      A     M 0.0;
      =     L 1.7;
      BLD   103;
      A     M 0.0;
      =     L 2.0;
      BLD   103;
      CALL  "FC_Auto_Reczny" (
           Enable                   := L 1.0,
           Reczny                   := L 1.1,
           Auto                     := L 1.2,
           Strefa_Bezp              := L 1.3,
           Test_Lampek              := L 1.4,
           Stop                     := L 1.5,
           Reset_1                  := L 1.6,
           Reset_2                  := L 1.7,
           Reset_3                  := L 2.0,
           Lampka_Reczny            := M 122.3,
           Lampka_Auto              := M 122.4,
           Auto_Reczny              := M 120.0);
      NOP   0;
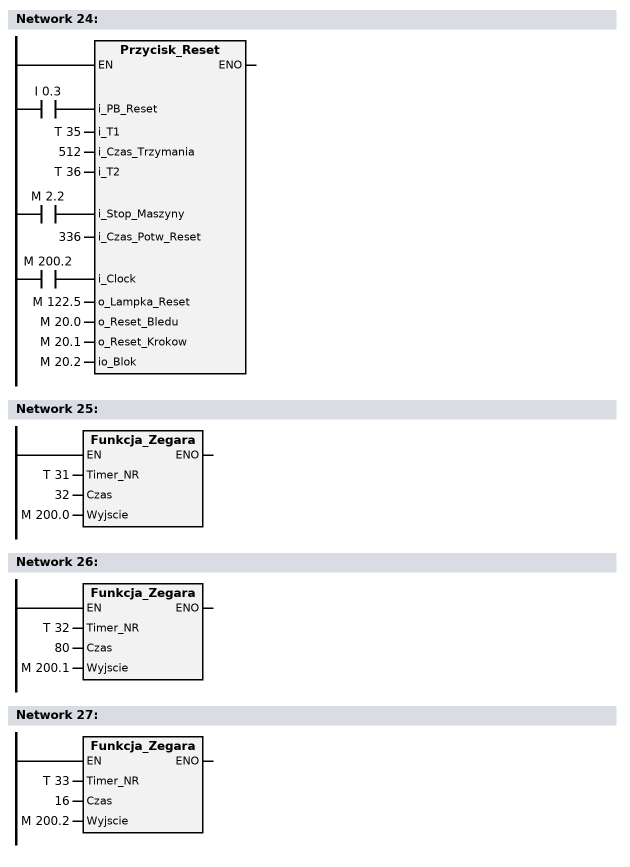
NETWORK
TITLE =
      A     I 0.3;
      =     L 1.0;
      BLD   103;
      A     M 2.2;
      =     L 1.1;
      BLD   103;
      A     M 200.2;
      =     L 1.2;
      BLD   103;
      CALL  "Przycisk_Reset" (
           i_PB_Reset               := L 1.0,
           i_T1                     := T 35,
           i_Czas_Trzymania         := 512,
           i_T2                     := T 36,
           i_Stop_Maszyny           := L 1.1,
           i_Czas_Potw_Reset        := 336,
           i_Clock                  := L 1.2,
           o_Lampka_Reset           := M 122.5,
           o_Reset_Bledu            := M 20.0,
           o_Reset_Krokow           := M 20.1,
           io_Blok                  := M 20.2);
      NOP   0;
NETWORK
TITLE =
//Timmer generujacy takt 200ms
//
      CALL  "Funkcja_Zegara" (
           Timer_NR                 := T 31,
           Czas                     := 32,
           Wyjscie                  := M 200.0);
      NOP   0;
NETWORK
TITLE =
//Timmer generujacy takt 500ms
      CALL  "Funkcja_Zegara" (
           Timer_NR                 := T 32,
           Czas                     := 80,
           Wyjscie                  := M 200.1);
      NOP   0;
NETWORK
TITLE =
//Timmer generujacy takt 100ms
      CALL  "Funkcja_Zegara" (
           Timer_NR                 := T 33,
           Czas                     := 16,
           Wyjscie                  := M 200.2);
      NOP   0;
END_FUNCTION

FUNCTION "Sprawdzenie_Czujnikow" : VOID	// FC 4
VERSION : 0.1
VAR_TEMP
  Help_Zmiana_1 : BOOL ;
  Help_Zmiana_2 : BOOL ;
  Help_Zmiana_3 : BOOL ;
  Help_Zmiana_4 : BOOL ;
END_VAR
BEGIN
NETWORK
TITLE =
//Ten Network celowo wolny
NETWORK
TITLE =
//Wyznaczenie zmian
//      A     "AIO".Banda_1.Foto_1
//      =     M    400.0
//      A     "AIO".Banda_2.Foto_1
//      =     M    400.1
      A     "AIO".Banda_3.Foto_1;
      =     M 400.2;
      A     "AIO".Banda_4.Foto_1;
      =     M 400.3;
      A     "AIO".Banda_4.Foto_2;
      =     M 400.4;
      A     "AIO".Banda_5.Foto_1;
      =     M 400.5;
      A     "AIO".Banda_6.Foto_1;
      =     M 400.6;
      A     "AIO".Banda_7.Foto_1;
      =     M 400.7;
      A     "AIO".Banda_8.Foto_1;
      =     M 401.0;
      A     "AIO".Banda_9.Foto_1;
      =     M 401.1;
      A     "AIO".Banda_10.Foto_1;
      =     M 401.2;
      A     "AIO".Banda_11.Foto_1;
      =     M 401.3;
      A     "AIO".Banda_12.Foto_1;
      =     M 401.4;
      A     "AIO".Banda_13.Foto_1;
      =     M 401.5;
      A     "AIO".Banda_13.Foto_2;
      =     M 401.6;
      A     "AIO".Banda_14.Foto_1;
      =     M 401.7;
      A     "AIO".Czuj_19.Czujnik_0_St;
      =     M 402.0;
      A     "AIO".Czuj_19.Czujnik_Ham_0_St;
      =     M 402.1;
      A     "AIO".Czuj_19.Czujnik_Ham_90_St;
      =     M 402.2;
      A     "AIO".Czuj_19.Czujnik_90_St;
      =     M 402.3;
      A     "AIO".Czuj_21.Czujnik_0_St;
      =     M 402.4;
      A     "AIO".Czuj_21.Czujnik_Ham_0_St;
      =     M 22.5;
      A     "AIO".Czuj_21.Czujnik_Ham_90_St;
      =     M 402.6;
      A     "AIO".Czuj_21.Czujnik_90_St;
      =     M 402.7;
      A     "AIO".Czuj_22.Czujnik_45_St_CW;
      =     M 403.0;
      A     "AIO".Czuj_22.Czujnik_45_St_CCW;
      =     M 403.1;
      A     "AIO".Banda_10.Foto_2;
      =     M 403.2;
//Czujnik od czesci bindujacej
      A     "AIO".Banda_23.Foto_1;
      =     M 408.0;
      A     "AIO".Banda_23.Foto_2;
      =     M 408.1;
      A     "AIO".Banda_24.Foto_1;
      =     M 408.2;
      A     "AIO".Banda_24.Foto_2;
      =     M 408.3;
      A     "AIO".Banda_2.Foto_1;
      =     M 408.4;
      A     "AIO".Banda_2.Foto_2;
      =     M 408.5;
//banda 1 wyjatkowo nie ma fotokomorek
//zamiast niej ma obrotnica 15
      A     "AIO".Obr_15.Foto_1;
      =     M 408.6;
      A     "AIO".Obr_15.Foto_2;
      =     M 408.7;
//-
      A     "AIO".Czuj_19_B.Czujnik_0_St;
      =     M 409.0;
      A     "AIO".Czuj_19_B.Czujnik_Ham_0_St;
      =     M 409.1;
      A     "AIO".Czuj_19_B.Czujnik_Ham_90_St;
      =     M 409.2;
      A     "AIO".Czuj_19_B.Czujnik_90_St;
      =     M 409.3;
//-
      A     "AIO".Czuj_17_B.Czujnik_180_St;
      =     M 409.4;
      A     "AIO".Czuj_17_B.Czujnik_Ham_180_St;
      =     M 409.5;
      A     "AIO".Czuj_17_B.Czujnik_Ham_270_St;
      =     M 409.6;
      A     "AIO".Czuj_17_B.Czujnik_270_St;
      =     M 409.7;
      A     I 2.7;
      =     M 410.0;
NETWORK
TITLE =
//pierwsze 32 bity do porownania
      CALL  "Szukaj_Zmiany_2" (
           DWORD_IN_NEW             := MD 400,
           CHANGE                   := #Help_Zmiana_1,
           DWORD_IN_OLD             := MD 404);
NETWORK
TITLE =
//drugie 32 bity do porownania
      CALL  "Szukaj_Zmiany_2" (
           DWORD_IN_NEW             := MD 408,
           CHANGE                   := #Help_Zmiana_2,
           DWORD_IN_OLD             := MD 412);
NETWORK
TITLE =
      CALL  "Toggle" (
           Wyzwolenie_1             := #Help_Zmiana_1,
           Wyzwolenie_2             := #Help_Zmiana_2,
           Wyzwolenie_3             := M 0.1,
           Wyzwolenie_4             := M 0.1,
           TOGGLE                   := M 5.0);
NETWORK
TITLE =
      A     M 5.0;
      =     M 123.1;
END_FUNCTION

FUNCTION "FC_Lampki" : VOID	// FC 6
VERSION : 0.1
VAR_INPUT
  in_0 : BOOL ;
  in_1 : BOOL ;
  in_2 : BOOL ;
  in_3 : BOOL ;
  in_4 : BOOL ;
  in_5 : BOOL ;
  in_6 : BOOL ;
  in_7 : BOOL ;
  Test : BOOL ;
END_VAR
VAR_OUTPUT
  out_0 : BOOL ;
  out_1 : BOOL ;
  out_2 : BOOL ;
  out_3 : BOOL ;
  out_4 : BOOL ;
  out_5 : BOOL ;
  out_6 : BOOL ;
  out_7 : BOOL ;
END_VAR
BEGIN
NETWORK
TITLE =
//przyporzadkowanie wejsc do wyjs
//0
      O     #in_0;
      O     #Test;
      =     #out_0;
//1
      O     #in_1;
      O     #Test;
      =     #out_1;
//2
      O     #in_2;
      O     #Test;
      =     #out_2;
//3
      O     #in_3;
      O     #Test;
      =     #out_3;
//4
      O     #in_4;
      O     #Test;
      =     #out_4;
//5
      O     #in_5;
      O     #Test;
      =     #out_5;
//6
      O     #in_6;
      O     #Test;
      =     #out_6;
//7
      O     #in_7;
      O     #Test;
      =     #out_7;
END_FUNCTION

FUNCTION "Szukaj_Zmiany_2" : VOID	// FC 7
//Funkcja wykrywa zmiane w obszarze wejscie i zapamietuje. Umozliwia to wykrycie 
//zmiany stanu kazdego czujnika lini. Funkcja ograniczona jest do dlugosci 32 
//bitow.
//
//Wersja 1.0
//Rozszerzenie dzia³ania funcji do 8 bajtow
AUTHOR : Kng
NAME : Help_FC
VERSION : 0.1
VAR_INPUT
  DWORD_IN_NEW : DWORD ;
END_VAR
VAR_OUTPUT
  CHANGE : BOOL ;
END_VAR
VAR_IN_OUT
  DWORD_IN_OLD : DWORD ;
END_VAR
BEGIN
NETWORK
TITLE =
//Sprawdz czy nastapila zmiana
      L     #DWORD_IN_NEW;
      L     #DWORD_IN_OLD;
      XOD;
      L     L#0;
      <>D;
      =     #CHANGE;
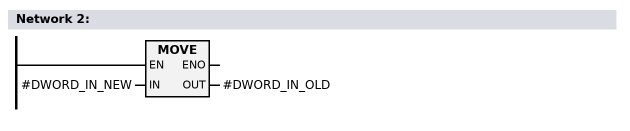
NETWORK
TITLE =
//Przypisz wartosc obecna jako stara
      L     #DWORD_IN_NEW;
      T     #DWORD_IN_OLD;
END_FUNCTION

FUNCTION "Toggle" : VOID	// FC 8
//Funcja zmienia stan wyjscia gdy ktore kolwiek wejscie zostanie wyzwolone
AUTHOR : Kng
NAME : Help_FC
VERSION : 0.1
VAR_INPUT
  Wyzwolenie_1 : BOOL ;
  Wyzwolenie_2 : BOOL ;
  Wyzwolenie_3 : BOOL ;
  Wyzwolenie_4 : BOOL ;
END_VAR
VAR_IN_OUT
  TOGGLE : BOOL ;
END_VAR
VAR_TEMP
  Temp_Bit_2 : BOOL ;
END_VAR
BEGIN
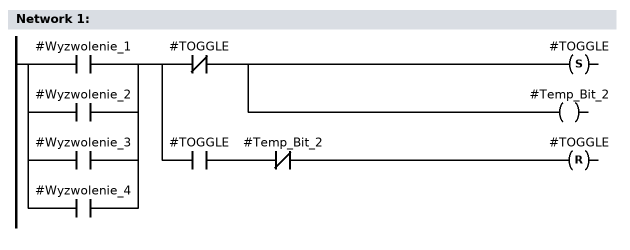
NETWORK
TITLE =
//Zapisz wykryta zminane
      O     #Wyzwolenie_1;
      O     #Wyzwolenie_2;
      O     #Wyzwolenie_3;
      O     #Wyzwolenie_4;
      =     L 1.0;
      A     L 1.0;
      AN    #TOGGLE;
      S     #TOGGLE;
      =     #Temp_Bit_2;
      A     L 1.0;
      A     #TOGGLE;
      AN    #Temp_Bit_2;
      R     #TOGGLE;
END_FUNCTION

FUNCTION "Sterwanie_Swiatlo" : VOID	// FC 9
VERSION : 0.1
VAR_TEMP
  Help_Bit : BOOL ;
END_VAR
BEGIN
NETWORK
TITLE =
//Ten Network celowo jest wolny
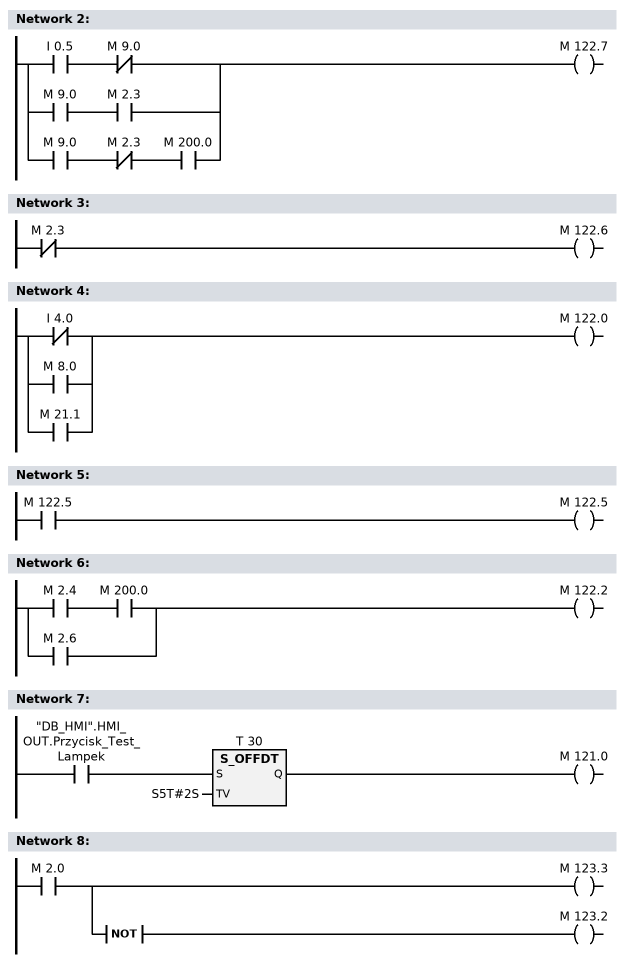
NETWORK
TITLE =
//Lampka pb start cyklu
      A     I 0.5;
      AN    M 9.0;
      O;
      A     M 9.0;
      A     M 2.3;
      O;
      A     M 9.0;
      AN    M 2.3;
      A     M 200.0;
      =     M 122.7;
NETWORK
TITLE =
//Lampka stop
      AN    M 2.3;
      =     M 122.6;
NETWORK
TITLE =
      ON    I 4.0;
      O     M 8.0;
      O     M 21.1;
      =     M 122.0;
NETWORK
TITLE =
//Miga reset
      A     M 122.5;
      =     M 122.5;
NETWORK
TITLE =
//Lampka bezpieczenstwa strefa
      A     M 2.4;
      A     M 200.0;
      O     M 2.6;
      =     M 122.2;
NETWORK
TITLE =
//Test Lampek z timmerem przedluzonym
      A     "DB_HMI".HMI_OUT.Przycisk_Test_Lampek;
      L     S5T#2S;
      SF    T 30;
      NOP   0;
      NOP   0;
      NOP   0;
      A     T 30;
      =     M 121.0;
NETWORK
TITLE =
//linia pracuje
      A     M 2.0;
      =     L 1.0;
      A     L 1.0;
      BLD   102;
      =     M 123.3;
      A     L 1.0;
      NOT;
      =     M 123.2;
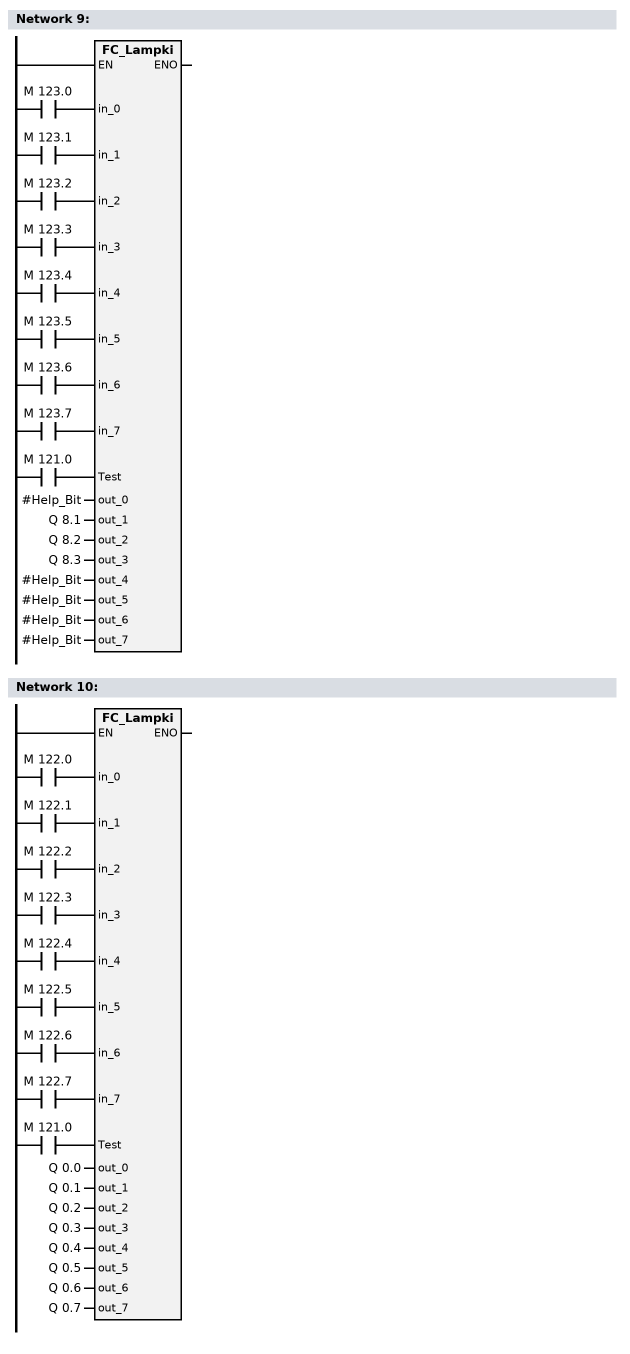
NETWORK
TITLE =
//Lampki na szafie sterowniczej sa troche przesuniete bo brakuje zielonej
      A     M 123.0;
      =     L 1.0;
      BLD   103;
      A     M 123.1;
      =     L 1.1;
      BLD   103;
      A     M 123.2;
      =     L 1.2;
      BLD   103;
      A     M 123.3;
      =     L 1.3;
      BLD   103;
      A     M 123.4;
      =     L 1.4;
      BLD   103;
      A     M 123.5;
      =     L 1.5;
      BLD   103;
      A     M 123.6;
      =     L 1.6;
      BLD   103;
      A     M 123.7;
      =     L 1.7;
      BLD   103;
      A     M 121.0;
      =     L 2.0;
      BLD   103;
      CALL  "FC_Lampki" (
           in_0                     := L 1.0,
           in_1                     := L 1.1,
           in_2                     := L 1.2,
           in_3                     := L 1.3,
           in_4                     := L 1.4,
           in_5                     := L 1.5,
           in_6                     := L 1.6,
           in_7                     := L 1.7,
           Test                     := L 2.0,
           out_0                    := #Help_Bit,
           out_1                    := Q 8.1,
           out_2                    := Q 8.2,
           out_3                    := Q 8.3,
           out_4                    := #Help_Bit,
           out_5                    := #Help_Bit,
           out_6                    := #Help_Bit,
           out_7                    := #Help_Bit);
      NOP   0;
NETWORK
TITLE =
//funkcja zarzadzajaca lampami
//Lampki na panelu operatorskim
      A     M 122.0;
      =     L 1.0;
      BLD   103;
      A     M 122.1;
      =     L 1.1;
      BLD   103;
      A     M 122.2;
      =     L 1.2;
      BLD   103;
      A     M 122.3;
      =     L 1.3;
      BLD   103;
      A     M 122.4;
      =     L 1.4;
      BLD   103;
      A     M 122.5;
      =     L 1.5;
      BLD   103;
      A     M 122.6;
      =     L 1.6;
      BLD   103;
      A     M 122.7;
      =     L 1.7;
      BLD   103;
      A     M 121.0;
      =     L 2.0;
      BLD   103;
      CALL  "FC_Lampki" (
           in_0                     := L 1.0,
           in_1                     := L 1.1,
           in_2                     := L 1.2,
           in_3                     := L 1.3,
           in_4                     := L 1.4,
           in_5                     := L 1.5,
           in_6                     := L 1.6,
           in_7                     := L 1.7,
           Test                     := L 2.0,
           out_0                    := Q 0.0,
           out_1                    := Q 0.1,
           out_2                    := Q 0.2,
           out_3                    := Q 0.3,
           out_4                    := Q 0.4,
           out_5                    := Q 0.5,
           out_6                    := Q 0.6,
           out_7                    := Q 0.7);
      NOP   0;
END_FUNCTION

FUNCTION "Przyporzadkowanie_Wejsc" : VOID	// FC 20
//Pobranie z bloku db stanu wejsc sieci asi i przyporzadkowanie do odpowiedniego 
//urzadzenia lini.
//NW35-adresy B
//
//
//Opis sygnalow od bindownicy:
//banda 23, 24, 1, 2 tworza zestaw tasm maszyny bindujacej
//obr 15 to obrotnica bindownicy
//25,26- to kurtyny
//16-rygiel
//17-modul resetu
AUTHOR : Kng
NAME : Help_FC
VERSION : 0.1
VAR_TEMP
  Help_Bit_1 : BOOL ;
  Help_Bit_2 : BOOL ;
  Help_Word_1 : INT ;
  Help_Word_2 : INT ;
END_VAR
BEGIN
NETWORK
TITLE =
//Ten network celowo jest wolny
NETWORK
TITLE =
NETWORK
TITLE = Silnik ok
//Banda Adres 1
      A     "Asi_input".Adres_1_bit_0;
      O     M 0.0;	//dodane
      =     "AIO".Banda_1.Silnik_OK;
      A     "Asi_input".Adres_1_bit_1;
      =     "AIO".Banda_1.Rezerwa_Silnik;
      A     "Asi_input".Adres_1_bit_2;
      =     "AIO".Banda_1.Foto_1;
      A     "Asi_input".Adres_1_bit_3;
      =     "AIO".Banda_1.Foto_2;
NETWORK
TITLE = Silnik ok
//Banda Adres 2
      A     "Asi_input".Adres_2_bit_0;
      O     M 0.0;
      =     "AIO".Banda_2.Silnik_OK;
      A     "Asi_input".Adres_2_bit_1;
      =     "AIO".Banda_2.Rezerwa_Silnik;
      A     "Asi_input".Adres_2_bit_2;
      =     "AIO".Banda_2.Foto_1;
      A     "Asi_input".Adres_2_bit_3;
      =     "AIO".Banda_2.Foto_2;
NETWORK
TITLE = Silnik ok
//Banda Adres 3
      A     "Asi_input".Adres_3_bit_0;
      =     "AIO".Banda_3.Silnik_OK;
      A     "Asi_input".Adres_3_bit_1;
      =     "AIO".Banda_3.Rezerwa_Silnik;
      A     "Asi_input".Adres_3_bit_2;
      =     "AIO".Banda_3.Foto_1;
      A     "Asi_input".Adres_3_bit_3;
      =     "AIO".Banda_3.Foto_2;
NETWORK
TITLE = Silnik ok
//Banda Adres 4
      A     "Asi_input".Adres_4_bit_0;
      =     "AIO".Banda_4.Silnik_OK;
      A     "Asi_input".Adres_4_bit_1;
      =     "AIO".Banda_4.Rezerwa_Silnik;
      A     "Asi_input".Adres_4_bit_2;
      =     "AIO".Banda_4.Foto_1;
      A     "Asi_input".Adres_4_bit_3;
      =     "AIO".Banda_4.Foto_2;
NETWORK
TITLE = Silnik ok
//Banda Adres 5
      A     "Asi_input".Adres_5_bit_0;
      =     "AIO".Banda_5.Silnik_OK;
      A     "Asi_input".Adres_5_bit_1;
      =     "AIO".Banda_5.Rezerwa_Silnik;
      A     "Asi_input".Adres_5_bit_2;
      =     "AIO".Banda_5.Foto_1;
      A     "Asi_input".Adres_5_bit_3;
      =     "AIO".Banda_5.Foto_2;
NETWORK
TITLE = Silnik ok
//Banda Adres 6
      A     "Asi_input".Adres_6_bit_0;
      =     "AIO".Banda_6.Silnik_OK;
      A     "Asi_input".Adres_6_bit_1;
      =     "AIO".Banda_6.Rezerwa_Silnik;
      A     "Asi_input".Adres_6_bit_2;
      =     "AIO".Banda_6.Foto_1;
      A     "Asi_input".Adres_6_bit_3;
      =     "AIO".Banda_6.Foto_2;
NETWORK
TITLE = Silnik ok
//Banda Adres 7
      A     "Asi_input".Adres_7_bit_0;
      =     "AIO".Banda_7.Silnik_OK;
      A     "Asi_input".Adres_7_bit_1;
      =     "AIO".Banda_7.Rezerwa_Silnik;
      A     "Asi_input".Adres_7_bit_2;
      =     "AIO".Banda_7.Foto_1;
      A     "Asi_input".Adres_7_bit_3;
      =     "AIO".Banda_7.Foto_2;
NETWORK
TITLE = Silnik ok
//Banda Adres 8
      A     "Asi_input".Adres_8_bit_0;
      =     "AIO".Banda_8.Silnik_OK;
      A     "Asi_input".Adres_8_bit_1;
      =     "AIO".Banda_8.Rezerwa_Silnik;
      A     "Asi_input".Adres_8_bit_2;
      =     "AIO".Banda_8.Foto_1;
      A     "Asi_input".Adres_8_bit_3;
      =     "AIO".Banda_8.Foto_2;
NETWORK
TITLE = Silnik ok
//Banda Adres 9
      A     "Asi_input".Adres_9_bit_0;
      =     "AIO".Banda_9.Silnik_OK;
      A     "Asi_input".Adres_9_bit_1;
      =     "AIO".Banda_9.Rezerwa_Silnik;
      A     "Asi_input".Adres_9_bit_2;
      =     "AIO".Banda_9.Foto_1;
      A     "Asi_input".Adres_9_bit_3;
      =     "AIO".Banda_9.Foto_2;
//Info do foliarki o zajetosci lini
      A     "AIO".Banda_9.Foto_1;
      =     "MPI_GD".OUT.Foto_Banda_9;
//-
NETWORK
TITLE = Silnik ok
//Banda Adres 10.Banda nalezy do foliarki.
      A     "Asi_input".Adres_10_bit_0;
      =     "AIO".Banda_10.Silnik_OK;
      A     "Asi_input".Adres_10_bit_1;
      =     "AIO".Banda_10.Rezerwa_Silnik;
      A     "Asi_input".Adres_10_bit_2;
      =     "AIO".Banda_10.Foto_1;
      A     "Asi_input".Adres_10_bit_3;
      =     "AIO".Banda_10.Foto_2;
//Sygnaly do foliarki
      A     "AIO".Banda_10.Silnik_OK;
      =     "MPI_GD".OUT.Silnik_10_OK;
//-
      A     "AIO".Banda_10.Foto_1;
      =     "MPI_GD".OUT.Foto_1_Banda_10;
//-
      A     "AIO".Banda_10.Foto_2;
      =     "MPI_GD".OUT.Foto_2_Banda_10;
NETWORK
TITLE = Silnik ok
//Banda Adres 11. Banda nalezy do foliarki.
      A     "Asi_input".Adres_11_bit_0;
      =     "AIO".Banda_11.Silnik_OK;
      A     "Asi_input".Adres_11_bit_1;
      =     "AIO".Banda_11.Rezerwa_Silnik;
      A     "Asi_input".Adres_11_bit_2;
      =     "AIO".Banda_11.Foto_1;
      A     "Asi_input".Adres_11_bit_3;
      =     "AIO".Banda_11.Foto_2;
//Sygnaly do foliarki
      A     "AIO".Banda_11.Silnik_OK;
      =     "MPI_GD".OUT.Silnik_11_OK;
//-
      A     "AIO".Banda_11.Foto_1;
      =     "MPI_GD".OUT.Foto_Banda_11;
NETWORK
TITLE = Silnik ok
//Banda Adres 12
      A     "Asi_input".Adres_12_bit_0;
      =     "AIO".Banda_12.Silnik_OK;
      A     "Asi_input".Adres_12_bit_1;
      =     "AIO".Banda_12.Rezerwa_Silnik;
      A     "Asi_input".Adres_12_bit_2;
      =     "AIO".Banda_12.Foto_1;
      A     "Asi_input".Adres_12_bit_3;
      =     "AIO".Banda_12.Foto_2;
NETWORK
TITLE = Silnik ok
//Banda Adres 13
      A     "Asi_input".Adres_13_bit_0;
      =     "AIO".Banda_13.Silnik_OK;
      A     "Asi_input".Adres_13_bit_1;
      =     "AIO".Banda_13.Rezerwa_Silnik;
      A     "Asi_input".Adres_13_bit_2;
      =     "AIO".Banda_13.Foto_1;
      A     "Asi_input".Adres_13_bit_3;
      =     "AIO".Banda_13.Foto_2;
NETWORK
TITLE = Silnik ok
//Banda Adres 14
      A     "Asi_input".Adres_14_bit_0;
      =     "AIO".Banda_14.Silnik_OK;
      A     "Asi_input".Adres_14_bit_1;
      =     "AIO".Banda_14.Rezerwa_Silnik;
      A     "Asi_input".Adres_14_bit_2;
      =     "AIO".Banda_14.Foto_1;
      A     "Asi_input".Adres_14_bit_3;
      =     "AIO".Banda_14.Foto_2;
NETWORK
TITLE = Silnik ok
//Obrotnica Adres 15
      A     "Asi_input".Adres_15_bit_0;
      =     "AIO".Obr_15.Silnik_OK;
      A     "Asi_input".Adres_15_bit_1;
      =     "AIO".Obr_15.Rezerwa_Silnik;
      A     "Asi_input".Adres_15_bit_2;
      =     "AIO".Obr_15.Foto_1;
      A     "Asi_input".Adres_15_bit_3;
      =     "AIO".Obr_15.Foto_2;
NETWORK
TITLE = Silnik ok
//Uwaga modul safety !!!
//Rygiel Adres 16
      A     "Asi_input".Adres_16_bit_0;
      =     "AIO".Rygiel_16.OSSD_Tor_1_1;
      A     "Asi_input".Adres_16_bit_1;
      =     "AIO".Rygiel_16.OSSD_Tor_1_2;
      A     "Asi_input".Adres_16_bit_2;
      =     "AIO".Rygiel_16.OSSD_Tor_2_1;
      A     "Asi_input".Adres_16_bit_3;
      =     "AIO".Rygiel_16.OSSD_Tor_2_2;
NETWORK
TITLE = Silnik ok
//Reset kurtyn bezpieczenswa Adres 17
//Nie wykorzystywane wejscia
NETWORK
TITLE = Silnik ok
//Obrotnica Adres_18
      A     "Asi_input".Adres_18_bit_0;
      =     "AIO".Obr_18.Silnik_OK;
      A     "Asi_input".Adres_18_bit_1;
      =     "AIO".Obr_18.Rezerwa_Silnik;
      A     "Asi_input".Adres_18_bit_2;
      =     "AIO".Obr_18.Foto_1;
      A     "Asi_input".Adres_18_bit_3;
      =     "AIO".Obr_18.Foto_2;
NETWORK
TITLE = Silnik ok
//Czujniki obrotnicy 1 Adres 19
      A     "Asi_input".Adres_19_bit_0;
      =     "AIO".Czuj_19.Czujnik_0_St;
      A     "Asi_input".Adres_19_bit_1;
      =     "AIO".Czuj_19.Czujnik_Ham_0_St;
      A     "Asi_input".Adres_19_bit_2;
      =     "AIO".Czuj_19.Czujnik_Ham_90_St;
      A     "Asi_input".Adres_19_bit_3;
      =     "AIO".Czuj_19.Czujnik_90_St;
NETWORK
TITLE = Silnik ok
//Obrotnica Adres 20
      A     "Asi_input".Adres_20_bit_0;
      =     "AIO".Obr_20.Silnik_OK;
      A     "Asi_input".Adres_20_bit_1;
      =     "AIO".Obr_20.Rezerwa_Silnik;
      A     "Asi_input".Adres_20_bit_2;
      =     "AIO".Obr_20.Foto_1;
      A     "Asi_input".Adres_20_bit_3;
      =     "AIO".Obr_20.Foto_2;
NETWORK
TITLE = Silnik ok
//Czujniki Obrotnicy 2 Adres 21
      A     "Asi_input".Adres_21_bit_0;
      =     "AIO".Czuj_21.Czujnik_0_St;
      A     "Asi_input".Adres_21_bit_1;
      =     "AIO".Czuj_21.Czujnik_Ham_0_St;
      A     "Asi_input".Adres_21_bit_2;
      =     "AIO".Czuj_21.Czujnik_Ham_90_St;
      A     "Asi_input".Adres_21_bit_3;
      =     "AIO".Czuj_21.Czujnik_90_St;
NETWORK
TITLE = Silnik ok
//Czujniki Obrotnicy 2 Adres 22
      A     "Asi_input".Adres_22_bit_0;
      =     "AIO".Czuj_22.Czujnik_45_St_CW;
      A     "Asi_input".Adres_22_bit_1;
      =     "AIO".Czuj_22.Czujnik_45_St_CCW;
      A     "Asi_input".Adres_22_bit_2;
      =     "AIO".Czuj_22.Rez_0_2;
      A     "Asi_input".Adres_22_bit_3;
      =     "AIO".Czuj_22.Rez_0_3;
NETWORK
TITLE = Wejscie SEW 1
//Banda 23 znajdujaca sie bedaca banda wjazdowa do bindownicy
      A     "Asi_input".Adres_23_bit_0;
      =     "AIO".Banda_23.Silnik_OK;
      A     "Asi_input".Adres_23_bit_1;
      =     "AIO".Banda_23.Rezerwa_Silnik;
      A     "Asi_input".Adres_23_bit_2;
      =     "AIO".Banda_23.Foto_1;
      A     "Asi_input".Adres_23_bit_3;
      =     "AIO".Banda_23.Foto_2;
NETWORK
TITLE = Silnik ok
//Banda 24
      A     "Asi_input".Adres_24_bit_0;
      =     "AIO".Banda_24.Silnik_OK;
      A     "Asi_input".Adres_24_bit_1;
      =     "AIO".Banda_24.Rezerwa_Silnik;
      A     "Asi_input".Adres_24_bit_2;
      =     "AIO".Banda_24.Foto_1;
      A     "Asi_input".Adres_24_bit_3;
      =     "AIO".Banda_24.Foto_2;
NETWORK
TITLE =
//Sprawdzenie czujnikow Bezpieczenstwa lini
//Kurtyna 25
      A     "Asi_input".Adres_25_bit_0;
      =     "AIO".Kurtyna_25.OSSD_Tor_1_1;
      A     "Asi_input".Adres_25_bit_1;
      =     "AIO".Kurtyna_25.OSSD_Tor_1_2;
      A     "Asi_input".Adres_25_bit_2;
      =     "AIO".Kurtyna_25.OSSD_Tor_2_1;
      A     "Asi_input".Adres_25_bit_3;
      =     "AIO".Kurtyna_25.OSSD_Tor_2_2;
NETWORK
TITLE =
//Sprawdzenie czujnikow Bezpieczenstwa lini
//Kurtyna 26
      A     "Asi_input".Adres_26_bit_0;
      =     "AIO".Kurtyna_26.OSSD_Tor_1_1;
      A     "Asi_input".Adres_26_bit_1;
      =     "AIO".Kurtyna_26.OSSD_Tor_1_2;
      A     "Asi_input".Adres_26_bit_2;
      =     "AIO".Kurtyna_26.OSSD_Tor_2_1;
      A     "Asi_input".Adres_26_bit_3;
      =     "AIO".Kurtyna_26.OSSD_Tor_2_2;
NETWORK
TITLE = Silnik ok
//Sprawdzenie czujnikow Bezpieczenstwa lini
//Not Aus 27
      A     "Asi_input".Adres_27_bit_0;
      =     "AIO".ESTOP_27.EStop_Tor_1_1;
      A     "Asi_input".Adres_27_bit_1;
      =     "AIO".ESTOP_27.EStop_Tor_1_2;
      A     "Asi_input".Adres_27_bit_2;
      =     "AIO".ESTOP_27.EStop_Tor_2_1;
      A     "Asi_input".Adres_27_bit_3;
      =     "AIO".ESTOP_27.EStop_Tor_2_2;
NETWORK
TITLE =
//Sprawdzenie czujnikow Bezpieczenstwa lini
//Not Aus 28
      A     "Asi_input".Adres_28_bit_0;
      =     "AIO".ESTOP_28.EStop_Tor_1_1;
      A     "Asi_input".Adres_28_bit_1;
      =     "AIO".ESTOP_28.EStop_Tor_1_2;
      A     "Asi_input".Adres_28_bit_2;
      =     "AIO".ESTOP_28.EStop_Tor_2_1;
      A     "Asi_input".Adres_28_bit_3;
      =     "AIO".ESTOP_28.EStop_Tor_2_2;
NETWORK
TITLE =
//Sprawdzenie czujnikow Bezpieczenstwa lini
//Not Aus 29
      A     "Asi_input".Adres_29_bit_0;
      =     "AIO".ESTOP_29.EStop_Tor_1_1;
      A     "Asi_input".Adres_29_bit_1;
      =     "AIO".ESTOP_29.EStop_Tor_1_2;
      A     "Asi_input".Adres_29_bit_2;
      =     "AIO".ESTOP_29.EStop_Tor_2_1;
      A     "Asi_input".Adres_29_bit_3;
      =     "AIO".ESTOP_29.EStop_Tor_2_2;
NETWORK
TITLE =
//Sprawdzenie czujnikow Bezpieczenstwa lini
//Not Aus 30
      A     "Asi_input".Adres_30_bit_0;
      =     "AIO".ESTOP_30.EStop_Tor_1_1;
      A     "Asi_input".Adres_30_bit_1;
      =     "AIO".ESTOP_30.EStop_Tor_1_2;
      A     "Asi_input".Adres_30_bit_2;
      =     "AIO".ESTOP_30.EStop_Tor_2_1;
      A     "Asi_input".Adres_30_bit_3;
      =     "AIO".ESTOP_30.EStop_Tor_2_2;
NETWORK
TITLE =
//Sprawdzenie czujnikow Bezpieczenstwa lini
//Not Aus 31
      A     "Asi_input".Adres_31_bit_0;
      =     "AIO".ESTOP_31.EStop_Tor_1_1;
      A     "Asi_input".Adres_31_bit_1;
      =     "AIO".ESTOP_31.EStop_Tor_1_2;
      A     "Asi_input".Adres_31_bit_2;
      =     "AIO".ESTOP_31.EStop_Tor_2_1;
      A     "Asi_input".Adres_31_bit_3;
      =     "AIO".ESTOP_31.EStop_Tor_2_2;
NETWORK
TITLE =
//Segment adresow B
//Dotyczy jedynie bialych modulow inuput nie zawartych wyzej
NETWORK
TITLE =
//Czujnik bindownicy Adres 19B 
      A     "Asi_input".B_Adres_19_bit_0;
      =     "AIO".Czuj_19_B.Czujnik_0_St;
      A     "Asi_input".B_Adres_19_bit_1;
      =     "AIO".Czuj_19_B.Czujnik_Ham_0_St;
      A     "Asi_input".B_Adres_19_bit_2;
      =     "AIO".Czuj_19_B.Czujnik_Ham_90_St;
      A     "Asi_input".B_Adres_19_bit_3;
      =     "AIO".Czuj_19_B.Czujnik_90_St;
NETWORK
TITLE =
//Czujnik bindownicy Adres 17B 
      A     "Asi_input".B_Adres_17_bit_0;
      =     "AIO".Czuj_17_B.Czujnik_Ham_180_St;
      A     "Asi_input".B_Adres_17_bit_1;
      =     "AIO".Czuj_17_B.Czujnik_180_St;
      A     "Asi_input".B_Adres_17_bit_2;
      =     "AIO".Czuj_17_B.Czujnik_Ham_270_St;
      A     "Asi_input".B_Adres_17_bit_3;
      =     "AIO".Czuj_17_B.Czujnik_270_St;
END_FUNCTION

FUNCTION "Przyporzadkowanie_Wyjsc" : VOID	// FC 21
VERSION : 0.1
VAR_TEMP
  Temp_Word_1 : INT ;
  Help_Bit_1 : BOOL ;
END_VAR
BEGIN
NETWORK
TITLE =
//Ten Network celowo jest wolny
NETWORK
TITLE = Temporary placeholder variable
//Banda 1 Adres 1
//****************ClockWise*******************
      A     "AIO".Banda_1.CC_Wise;	//C_Wise
      =     "Asi_output".Adres_1_bit_0;
//****************CounterClockWise************
      A     "AIO".Banda_1.C_Wise;
      =     "Asi_output".Adres_1_bit_1;	//CC_Wise
//****************Wolno***********************
      A     "AIO".Banda_1.Wolno;
      O     I 0.0;
      =     "Asi_output".Adres_1_bit_2;	//Wolno
//****************Bit_Bezpieczenstwa**********
      A     M 2.0;	//Safety
      =     "Asi_output".Adres_1_bit_3;
NETWORK
TITLE = Temporary placeholder variable
//Banda 2 Adres 2
//****************ClockWise*******************
      A     "AIO".Banda_2.CC_Wise;	//C_Wise
      =     "Asi_output".Adres_2_bit_0;
//****************CounterClockWise************
      A     "AIO".Banda_2.C_Wise;
      =     "Asi_output".Adres_2_bit_1;	//CC_Wise
//****************Wolno***********************
      AN    "AIO".Banda_2.Wolno;
      =     "Asi_output".Adres_2_bit_2;	//Wolno
//****************Bit_Bezpieczenstwa**********
      A     M 2.0;	//Safety
      =     "Asi_output".Adres_2_bit_3;
NETWORK
TITLE = Temporary placeholder variable
//Banda 3 Adres 3
//****************ClockWise*******************
      A     M 0.1;	//C_Wise
      =     "Asi_output".Adres_3_bit_0;
//****************CounterClockWise************
      A     "AIO".Banda_3.C_Wise;
      =     "Asi_output".Adres_3_bit_1;	//CC_Wise
//****************Wolno***********************
      A     M 0.0;
      =     "Asi_output".Adres_3_bit_2;	//Wolno
//****************Bit_Bezpieczenstwa**********
      A     M 2.0;	//Safety
      =     "Asi_output".Adres_3_bit_3;
NETWORK
TITLE = Temporary placeholder variable
//Banda 4 Obrotnica
//****************ClockWise*******************
      A     "AIO".Banda_4.C_Wise;	//C_Wise
      =     "Asi_output".Adres_4_bit_0;
//****************CounterClockWise************
      A     "AIO".Banda_4.CC_Wise;
      =     "Asi_output".Adres_4_bit_1;	//CC_Wise
//****************Wolno***********************
      A     M 0.0;
      =     "Asi_output".Adres_4_bit_2;	//Wolno
//****************Bit_Bezpieczenstwa**********
      A     M 2.0;	//Safety
      =     "Asi_output".Adres_4_bit_3;
NETWORK
TITLE = Temporary placeholder variable
//Banda 5 Rolki
//****************ClockWise*******************
      A     M 0.1;	//C_Wise
      =     "Asi_output".Adres_5_bit_0;
//****************CounterClockWise************
      A     "AIO".Banda_5.C_Wise;
      =     "Asi_output".Adres_5_bit_1;	//CC_Wise
//****************Wolno***********************
      A     M 0.0;
      =     "Asi_output".Adres_5_bit_2;	//Wolno
//****************Bit_Bezpieczenstwa**********
      A     M 2.0;	//Safety
      =     "Asi_output".Adres_5_bit_3;
NETWORK
TITLE = Temporary placeholder variable
//Banda 6 Rolki
//****************ClockWise*******************
      A     "AIO".Banda_6.C_Wise;	//C_Wise
      =     "Asi_output".Adres_6_bit_0;
//****************CounterClockWise************
      A     M 0.1;
      =     "Asi_output".Adres_6_bit_1;	//CC_Wise
//****************Wolno***********************
      A     M 0.1;
      =     "Asi_output".Adres_6_bit_2;	//Wolno
//****************Bit_Bezpieczenstwa**********
      A     M 2.0;	//Safety
      =     "Asi_output".Adres_6_bit_3;
NETWORK
TITLE = Temporary placeholder variable
//Banda 7 Rolki
//****************ClockWise*******************
      A     M 0.1;	//C_Wise
      =     "Asi_output".Adres_7_bit_0;
//****************CounterClockWise************
      A     "AIO".Banda_7.C_Wise;
      =     "Asi_output".Adres_7_bit_1;	//CC_Wise
//****************Wolno***********************
      A     M 0.0;
      =     "Asi_output".Adres_7_bit_2;	//Wolno
//****************Bit_Bezpieczenstwa**********
      A     M 2.0;	//Safety
      =     "Asi_output".Adres_7_bit_3;
NETWORK
TITLE = Temporary placeholder variable
//Banda 8 Rolki
//****************ClockWise*******************
      A     "AIO".Banda_8.C_Wise;	//C_Wise
      =     "Asi_output".Adres_8_bit_0;
//****************CounterClockWise************
      A     M 0.1;
      =     "Asi_output".Adres_8_bit_1;	//CC_Wise
//****************Wolno***********************
      A     M 0.1;
      =     "Asi_output".Adres_8_bit_2;	//Wolno
//****************Bit_Bezpieczenstwa**********
      A     M 2.0;	//Safety
      =     "Asi_output".Adres_8_bit_3;
NETWORK
TITLE = Temporary placeholder variable
//Banda 9 Rolki
//****************ClockWise*******************
      A     M 0.1;	//C_Wise
      =     "Asi_output".Adres_9_bit_0;
//****************CounterClockWise************
      A     "AIO".Banda_9.C_Wise;
      =     "Asi_output".Adres_9_bit_1;	//CC_Wise
//****************Wolno***********************
      A     M 0.0;
      =     "Asi_output".Adres_9_bit_2;	//Wolno
//****************Bit_Bezpieczenstwa**********
      A     M 2.0;	//Safety
      =     "Asi_output".Adres_9_bit_3;
NETWORK
TITLE = Temporary placeholder variable
//Banda 10 Rolki
//Uwaga Banda ta nalezy do foliarki
//Sygnaly z foliarki
      A     "MPI_GD".IN.Motor_10_Lewo;
      =     "AIO".Banda_10.C_Wise;
      A     "MPI_GD".IN.Motor_10_Prawo;
      =     "AIO".Banda_10.CC_Wise;
//****************ClockWise*******************
      A     "AIO".Banda_10.C_Wise;	//C_Wise
      =     "Asi_output".Adres_10_bit_0;
//****************CounterClockWise************
      A     "AIO".Banda_10.CC_Wise;
      =     "Asi_output".Adres_10_bit_1;	//CC_Wise
//****************Wolno***********************
      A     M 0.0;
      =     "Asi_output".Adres_10_bit_2;	//Wolno
//****************Bit_Bezpieczenstwa**********
      A     M 2.0;	//Safety
      =     "Asi_output".Adres_10_bit_3;
NETWORK
TITLE = Temporary placeholder variable
//Banda 11 Rolki
//Uwaga Banda ta nalezy do foliarki
//Sygnaly z foliarki
      A     "MPI_GD".IN.Motor_11_Lewo;
      =     "AIO".Banda_11.C_Wise;
      A     "MPI_GD".IN.Motor_11_Prawo;
      =     "AIO".Banda_11.CC_Wise;
//****************ClockWise*******************
      A     "AIO".Banda_11.C_Wise;	//C_Wise
      =     "Asi_output".Adres_11_bit_0;
//****************CounterClockWise************
      A     "AIO".Banda_11.CC_Wise;
      =     "Asi_output".Adres_11_bit_1;	//CC_Wise
//****************Wolno***********************
      A     M 0.0;
      =     "Asi_output".Adres_11_bit_2;	//Wolno
//****************Bit_Bezpieczenstwa**********
      A     M 2.0;	//Safety
      =     "Asi_output".Adres_11_bit_3;
NETWORK
TITLE = Temporary placeholder variable
//Banda 12 Rolki wlot 2 na obrotnice
//****************ClockWise*******************
      A     "AIO".Banda_12.C_Wise;	//C_Wise
      =     "Asi_output".Adres_12_bit_0;
//****************CounterClockWise************
      A     M 0.1;
      =     "Asi_output".Adres_12_bit_1;	//CC_Wise
//****************Wolno***********************
      A     M 0.1;
      =     "Asi_output".Adres_12_bit_2;	//Wolno
//****************Bit_Bezpieczenstwa**********
      A     M 2.0;	//Safety
      =     "Asi_output".Adres_12_bit_3;
NETWORK
TITLE = Temporary placeholder variable
//Banda 13 Adres 13 Rolki na obrotnicy
//****************ClockWise*******************
      A     "AIO".Banda_13.C_Wise;	//C_Wise
      =     "Asi_output".Adres_13_bit_0;
//****************CounterClockWise************
      A     "AIO".Banda_13.CC_Wise;
      =     "Asi_output".Adres_13_bit_1;	//CC_Wise
//****************Wolno***********************
      A     M 0.1;
      =     "Asi_output".Adres_13_bit_2;	//Wolno
//****************Bit_Bezpieczenstwa**********
      A     M 2.0;	//Safety
      =     "Asi_output".Adres_13_bit_3;
NETWORK
TITLE = Temporary placeholder variable
//Banda 14 Adres 14 Wylot z maszyny
//****************ClockWise*******************
      A     "AIO".Banda_14.C_Wise;	//C_Wise
      =     "Asi_output".Adres_14_bit_0;
//****************CounterClockWise************
      A     M 0.1;
      =     "Asi_output".Adres_14_bit_1;	//CC_Wise
//****************Wolno***********************
      A     M 0.1;
      =     "Asi_output".Adres_14_bit_2;	//Wolno
//****************Bit_Bezpieczenstwa**********
      A     M 2.0;	//Safety
      =     "Asi_output".Adres_14_bit_3;
NETWORK
TITLE = Temporary placeholder variable
//Obrotnica 15 Adres 15
//****************ClockWise*******************
      A     "AIO".Obr_15.C_Wise;
      =     "Asi_output".Adres_15_bit_0;
//****************CounterClockWise************
      A     "AIO".Obr_15.CC_Wise;
      =     "Asi_output".Adres_15_bit_1;	//CC_Wise
//****************Wolno***********************
      AN    "AIO".Obr_15.Wolno;
      =     "Asi_output".Adres_15_bit_2;	//Wolno
//****************Bit_Bezpieczenstwa**********
      A     M 2.0;	//Safety
      =     "Asi_output".Adres_15_bit_3;
NETWORK
TITLE =
//adres 16 rygiel brak output
NETWORK
TITLE = Temporary placeholder variable
//adres 17 reset kurtyn
//****************Reset wlot *****************
      A     "AIO".Reset_17.Reset_Wlot;
      =     "Asi_output".Adres_17_bit_0;	//reset wlot
//****************Reset wylot ****************
      A     "AIO".Reset_17.Reset_Wylot;
      =     "Asi_output".Adres_17_bit_1;	//reset wylot
NETWORK
TITLE = Temporary placeholder variable
//Obrotnica 18  Adres 18
//****************ClockWise*******************
      A     "AIO".Obr_18.C_Wise;
      =     "Asi_output".Adres_18_bit_0;
//****************CounterClockWise************
      A     "AIO".Obr_18.CC_Wise;
      =     "Asi_output".Adres_18_bit_1;	//CC_Wise
//****************Wolno***********************
      A     "AIO".Obr_18.Wolno;
      =     "Asi_output".Adres_18_bit_2;	//Wolno
//****************Bit_Bezpieczenstwa**********
      A     M 2.0;	//Safety
      =     "Asi_output".Adres_18_bit_3;
NETWORK
TITLE = Temporary placeholder variable
//Adres 19 brak sygnalow output
NETWORK
TITLE = Temporary placeholder variable
//Obrotnica 20 Adres 20
//****************ClockWise*******************
      A     "AIO".Obr_20.C_Wise;
      =     "Asi_output".Adres_20_bit_0;
//****************CounterClockWise************
      A     "AIO".Obr_20.CC_Wise;
      =     "Asi_output".Adres_20_bit_1;	//CC_Wise
//****************Wolno***********************
      A     "AIO".Obr_20.Wolno;
      =     "Asi_output".Adres_20_bit_2;	//Wolno
//****************Bit_Bezpieczenstwa**********
      A     M 2.0;	//Safety
      =     "Asi_output".Adres_20_bit_3;
NETWORK
TITLE = Temporary placeholder variable
//Adres 21, 22 Brak Output
NETWORK
TITLE = Temporary placeholder variable
//Banda 23
//
//****************ClockWise*******************
      A     "AIO".Banda_23.CC_Wise;	//C_Wise
      =     "Asi_output".Adres_23_bit_0;
//****************CounterClockWise************
      A     "AIO".Banda_23.C_Wise;
      =     "Asi_output".Adres_23_bit_1;	//CC_Wise
//****************Wolno***********************
      A     "AIO".Banda_23.Wolno;
      =     "Asi_output".Adres_23_bit_2;	//Wolno
//****************Bit_Bezpieczenstwa**********
      A     M 2.0;	//Safety
      =     "Asi_output".Adres_23_bit_3;
NETWORK
TITLE = Temporary placeholder variable
//Banda 24
//
//****************ClockWise*******************
      A     "AIO".Banda_24.CC_Wise;	//C_Wise
      =     "Asi_output".Adres_24_bit_0;
//****************CounterClockWise************
      A     "AIO".Banda_24.C_Wise;
      =     "Asi_output".Adres_24_bit_1;	//CC_Wise
//****************Wolno***********************
      A     M 0.0;
      =     "Asi_output".Adres_24_bit_2;	//Wolno
//****************Bit_Bezpieczenstwa**********
      A     M 2.0;	//Safety
      =     "Asi_output".Adres_24_bit_3;
NETWORK
TITLE =
//25,26 to kurtyny bezpieczenstwa brak output
NETWORK
TITLE =
//Aedrs 27,28,29,30,31. Adresy ESTOP brak syganlow output
NETWORK
TITLE =
//Dziekuje za uwage
END_FUNCTION

FUNCTION "Rejestr_Tasm" : VOID	// FC 30
VERSION : 0.1
BEGIN
NETWORK
TITLE =
//marki uzywane od mb60. 
//Palety sa przekazywane za pomoca rejstru przesuwnego bitowego
//Poczatek monitorowania
      O     "AIO".Banda_4.Foto_1;
      O     "AIO".Banda_4.Foto_2;
      A     "AIO".Banda_4.Potw_Dost_Wlot_2;
      S     M 60.0;
//Przekazanie na pierwsza bande (banda 5)
      A     "AIO".Banda_5.Foto_1;
      A     "AIO".Banda_5.Paleta_Dost_do_Pop;
      A     M 60.0;
      JCN   et_1;
      S     M 60.1;
      R     M 60.0;
et_1: NOP   0;
      A     "AIO".Banda_6.Foto_1;
      A     "AIO".Banda_6.Paleta_Dost_do_Pop;
      A     M 60.1;
      JCN   et_2;
      S     M 60.2;
      R     M 60.1;
et_2: NOP   0;
      A     "AIO".Banda_7.Foto_1;
      A     "AIO".Banda_7.Paleta_Dost_do_Pop;
      A     M 60.2;
      JCN   et_3;
      S     M 60.3;
      R     M 60.2;
et_3: NOP   0;
      A     "AIO".Banda_8.Foto_1;
      A     "AIO".Banda_8.Paleta_Dost_do_Pop;
      A     M 60.3;
      JCN   et_4;
      S     M 60.4;
      R     M 60.3;
et_4: NOP   0;
      A     "AIO".Banda_9.Foto_1;
      A     "AIO".Banda_9.Paleta_Dost_do_Pop;
      A     M 60.4;
      JCN   et_5;
      S     M 60.5;
      R     M 60.4;
et_5: NOP   0;
//Banda 10 to foliarka
      A     "AIO".Banda_10.Foto_1;
      A     "AIO".Banda_10.Paleta_Dost_do_Pop;
      A     M 60.5;
      JCN   et_6;
      S     M 60.6;
      R     M 60.5;
et_6: NOP   0;
      A     M 60.6;
      A     "MPI_GD".IN.Foto_Banda_1;	// run in 
      S     M 62.0;
      A     M 62.0;
      A     "MPI_GD".IN.Foto_Owijarka;	//foto banda 4
      JCN   et_7;
      S     M 66.7;
      R     M 66.6;
      R     M 66.2;
et_7: NOP   0;
      A     M 66.7;
      =     "MPI_GD".OUT.Zmien_Program_Na_4;
      A     "MPI_GD".IN.Rezerwa_1;
      R     M 66.7;
//nie gotowe wiec wszystkie foliowane
      SET;
      R     "MPI_GD".OUT.Zmien_Program_Na_4;
      R     "MPI_GD".OUT.Zmien_Pragram_Na_3;
END_FUNCTION

FUNCTION "FC_Auto_Reczny" : VOID	// FC 40
//Funkcja przelaczajaca miedzy auto i recznym
VERSION : 0.1
VAR_INPUT
  Enable : BOOL ;	//Zezwolenie na dzia³anie
  Reczny : BOOL ;
  Auto : BOOL ;
  Strefa_Bezp : BOOL ;
  Test_Lampek : BOOL ;	//test lampek
  Stop : BOOL ;
  Reset_1 : BOOL ;
  Reset_2 : BOOL ;
  Reset_3 : BOOL ;
END_VAR
VAR_OUTPUT
  Lampka_Reczny : BOOL ;
  Lampka_Auto : BOOL ;
END_VAR
VAR_IN_OUT
  Auto_Reczny : BOOL ;	//Auto 1, Reczny 0
END_VAR
BEGIN
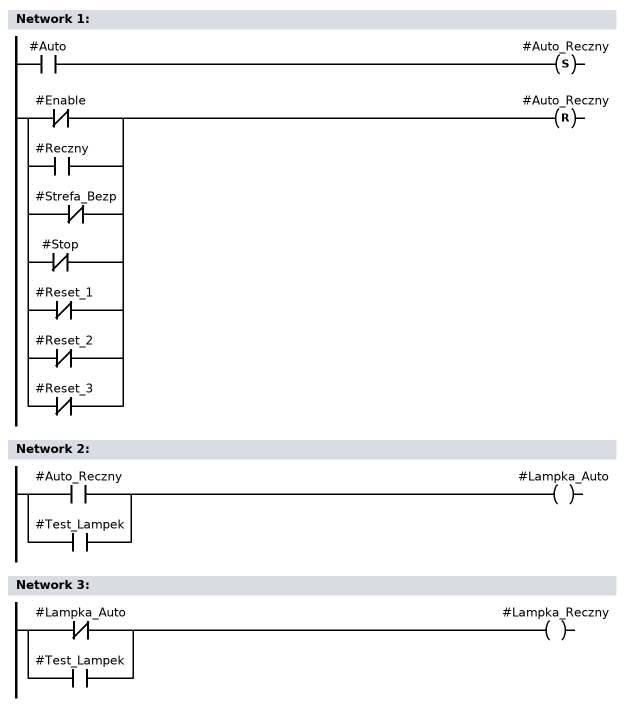
NETWORK
TITLE =
      A     #Auto;
      S     #Auto_Reczny;
      A(;
      ON    #Enable;
      O     #Reczny;
      ON    #Strefa_Bezp;
      ON    #Stop;
      ON    #Reset_1;
      ON    #Reset_2;
      ON    #Reset_3;
      );
      R     #Auto_Reczny;
      NOP   0;
NETWORK
TITLE =
      O     #Auto_Reczny;
      O     #Test_Lampek;
      =     #Lampka_Auto;
NETWORK
TITLE =
      ON    #Lampka_Auto;
      O     #Test_Lampek;
      =     #Lampka_Reczny;
END_FUNCTION

FUNCTION "Przycisk_Reset" : VOID	// FC 41
//Funkcja sluzy do jednoczesnej oblugi bledow oraz kasowania aktualnego kroku. 
//-Jezeli wcisnie sie przycisk to krotko do 5s to nastopi pruba kasowania bledu.
//-Jezeli wcisnie sie przycisk dlugo powyzej 5s to nastapi szybkie migniecie i 
//reset krokow
//
VERSION : 0.1
VAR_INPUT
  i_PB_Reset : BOOL ;
  i_T1 : TIMER ;	//Timer do dlugiego resetowania
  i_Czas_Trzymania : S5TIME ;
  i_T2 : TIMER ;	//Timer migania po przycisku
  i_Stop_Maszyny : BOOL ;
  i_Czas_Potw_Reset : S5TIME ;
  i_Clock : BOOL ;	//Zegar 100ms
END_VAR
VAR_OUTPUT
  o_Lampka_Reset : BOOL ;
END_VAR
VAR_IN_OUT
  o_Reset_Bledu : BOOL ;
  o_Reset_Krokow : BOOL ;
  io_Blok : BOOL ;
END_VAR
VAR_TEMP
  Temp_Help_1 : BOOL ;
  Temp_Help_2 : BOOL ;
END_VAR
BEGIN
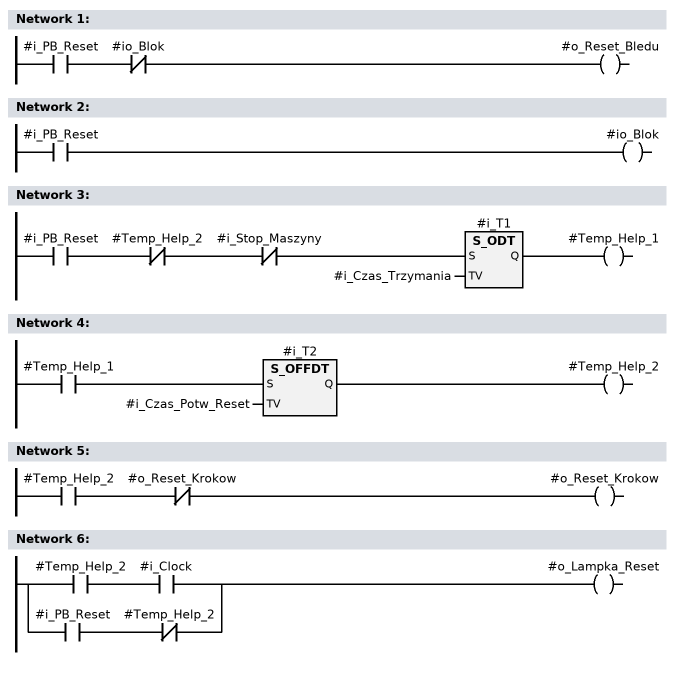
NETWORK
TITLE =
      A     #i_PB_Reset;
      AN    #io_Blok;
      =     #o_Reset_Bledu;
NETWORK
TITLE =
      A     #i_PB_Reset;
      =     #io_Blok;
NETWORK
TITLE =
      A     #i_PB_Reset;
      AN    #Temp_Help_2;
      AN    #i_Stop_Maszyny;
      L     #i_Czas_Trzymania;
      SD    #i_T1;
      NOP   0;
      NOP   0;
      NOP   0;
      A     #i_T1;
      =     #Temp_Help_1;
NETWORK
TITLE =
      A     #Temp_Help_1;
      L     #i_Czas_Potw_Reset;
      SF    #i_T2;
      NOP   0;
      NOP   0;
      NOP   0;
      A     #i_T2;
      =     #Temp_Help_2;
NETWORK
TITLE =
//Reset krokow
      A     #Temp_Help_2;
      AN    #o_Reset_Krokow;
      =     #o_Reset_Krokow;
NETWORK
TITLE =
//Lampka reset
      A     #Temp_Help_2;
      A     #i_Clock;
      O;
      A     #i_PB_Reset;
      AN    #Temp_Help_2;
      =     #o_Lampka_Reset;
END_FUNCTION

FUNCTION "ASI_Odczyt" : VOID	// FC 80
//Pobieranie danych z modulu ASI CP 342-2
AUTHOR : Kng
FAMILY : Asi_fun
NAME : r_ASi
VERSION : 0.1
VAR_INPUT
  CP_Adr : INT ;
  DB_Nr : INT ;
END_VAR
VAR_TEMP
  L_CP_Adr : DWORD ;
  L_DB_Target : WORD ;
  L_Start_Adr : DWORD ;
  L_Count : WORD ;
  Word_CP_Adr : WORD ;
  Fault : INT ;
  Target : ANY ;
END_VAR
BEGIN
NETWORK
TITLE =
      L     #CP_Adr;	// Adres urzadzenia
      SLD   3;	//Przejscie na wskaznik
      T     #L_CP_Adr;
      L     #DB_Nr;	// Nr bloku db
      T     #L_DB_Target;
      L     0;	// Start adres db 
      SLD   3;	// Przejscie na wskaznik
      T     #L_Start_Adr;
      L     4;	// Liczba petli (pobranie 16 bajtow)
next: T     #L_Count;
      L     PID [#L_CP_Adr];	// Zaladowanie wejsc
      OPN   DB [#L_DB_Target];	// Otwarcie db
      T     DBD [#L_Start_Adr];	// Wgranie danych
      L     #L_CP_Adr;	// Zaladuj adres cp
      SRD   3;	// przejscie na format obliczen
      L     4;
      +I;	// bo doble word 
      SLD   3;	// Przejscie na wskaznik
      T     #L_CP_Adr;
      L     #L_Start_Adr;	// Przesuniecie bloku danych
      SRD   3;	// do nastepnego ladowania
      L     4;
      +I;	// 
      SLD   3;	// 
      T     #L_Start_Adr;
      L     #L_Count;
      LOOP  next;	// powrot petli  next
NETWORK
TITLE =
//Recnum nie wiem co to jest dana z kart katologowych
//Funkcja ta odpowiada za segment adresowania B
      LAR1  P##Target;	// wskaznik do obszaru  docelowego
      L     W#16#1002;	//zaladuj skladnie 10 i typ byte 02
      T     LW [AR1,P#0.0];
      L     16;	//zaladuj dl. obszaru do kopiowania
      T     LW [AR1,P#2.0];
      L     #DB_Nr;	//zaladuj nr bloku db (np.:db33)
      T     LW [AR1,P#4.0];
      L     16;	//zaladuj start_adres odbioru danych
      SLD   3;	// przesun w lewo (bit ostatni ma 0.0
      OD    DW#16#84000000;	//ustaw wartosc 84-db
      T     LD [AR1,P#6.0];
//------------------------------------
      L     #CP_Adr;
      T     #Word_CP_Adr;
      CALL  "RD_REC" (
           REQ                      := TRUE,
           IOID                     := B#16#54,
           LADDR                    := #Word_CP_Adr,
           RECNUM                   := B#16#96,
           RET_VAL                  := #Fault,
           BUSY                     := L 16.1,
           RECORD                   := #Target);
END_FUNCTION

FUNCTION "ASI_Zapis" : VOID	// FC 81
//Wgranie danych do modulu ASI CP 342-2
//Funkcja ta powinna znalezc sie po programie przypiania wyjsc!!!!
AUTHOR : Kng
FAMILY : Asi_fun
NAME : w_ASi
VERSION : 0.1
VAR_INPUT
  CP_Adr : INT ;	//Adres modulu cp343-2
  DB_Nr : INT ;	//Nr db z ktorego pobierane dane
END_VAR
VAR_TEMP
  L_CP_Adr : DWORD ;
  L_DB_Target : WORD ;
  L_Start_Adr : DWORD ;
  L_Count : WORD ;
  Word_CP_Adr : WORD ;
  Fault : INT ;
  Source : ANY ;
END_VAR
BEGIN
NETWORK
TITLE =
      L     #CP_Adr;	// Adres urzadzenia
      SLD   3;	//Przejscie na wskaznik
      T     #L_CP_Adr;
      L     #DB_Nr;	// Nr bloku db
      T     #L_DB_Target;
      L     0;	// Start adres db 
      SLD   3;	// Przejscie na wskaznik
      T     #L_Start_Adr;
      L     4;	// Liczba petli (pobranie 16 bajtow)
next: T     #L_Count;
      OPN   DB [#L_DB_Target];	// Otwarcie db
      L     DBD [#L_Start_Adr];	// Zaladowanie danych
      T     PQD [#L_CP_Adr];	// Wgranie wyjsc
      L     #L_CP_Adr;	// Zaladuj adres cp
      SRD   3;	// przejscie na format obliczen
      L     4;
      +I;	// bo double word 
      SLD   3;	// Przejscie na wskaznik
      T     #L_CP_Adr;
      L     #L_Start_Adr;	// Przesuniecie bloku danych
      SRD   3;	// do nastepnego ladowania
      L     4;
      +I;	// 
      SLD   3;	// 
      T     #L_Start_Adr;
      L     #L_Count;
      LOOP  next;	// powrot petli  next
//mala maszyna to dodac beu
NETWORK
TITLE =
//Recnum nie wiem co to jest dana z kart katologowych
//Funkcja ta odpowiada za segment adresowania B
      LAR1  P##Source;	// wskaznik do obszaru  pobierajacego
      L     W#16#1002;	//zaladuj skladnie 10 i typ byte 02
      T     LW [AR1,P#0.0];
      L     16;	//zaladuj dl. obszaru do kopiowania
      T     LW [AR1,P#2.0];
      L     #DB_Nr;	//zaladuj nr bloku db (np.:db33)
      T     LW [AR1,P#4.0];
      L     16;	//zaladuj start_adres odbioru danych
      SLD   3;	// przesun w lewo (bit ostatni ma 0.0
      OD    DW#16#84000000;	//ustaw wartosc 84-db
      T     LD [AR1,P#6.0];
//------------------------------------
      L     #CP_Adr;
      T     #Word_CP_Adr;
      CALL  "WR_REC" (
           REQ                      := TRUE,
           IOID                     := B#16#55,
           LADDR                    := #Word_CP_Adr,
           RECNUM                   := B#16#96,
           RECORD                   := #Source,
           RET_VAL                  := #Fault,
           BUSY                     := L 16.1);
END_FUNCTION

FUNCTION "Opoznienie_Wylotu" : VOID	// FC 85
VERSION : 0.1
VAR_INPUT
  Wejscie : BOOL ;	//Fotokomorka
  Timmer_1 : TIMER ;
  Timmer_2 : TIMER ;
END_VAR
VAR_OUTPUT
  Wyjscie : BOOL ;
END_VAR
VAR_IN_OUT
  Zmienna : BOOL ;
END_VAR
BEGIN
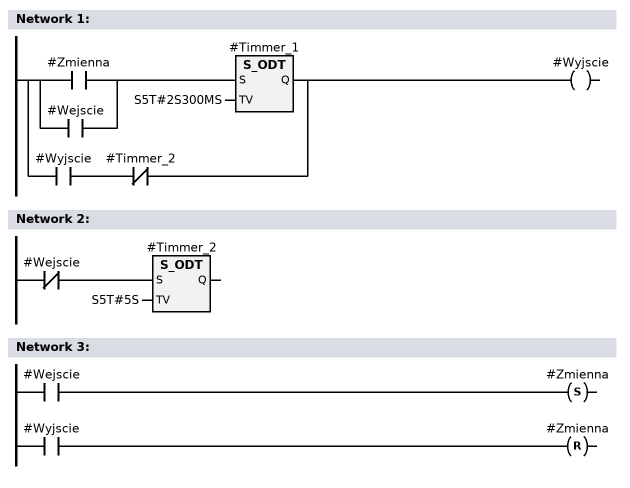
NETWORK
TITLE =
      O(;
      A(;
      O     #Zmienna;
      O     #Wejscie;
      );
      L     S5T#2S300MS;
      SD    #Timmer_1;
      NOP   0;
      NOP   0;
      NOP   0;
      A     #Timmer_1;
      );
      O;
      A     #Wyjscie;
      AN    #Timmer_2;
      =     #Wyjscie;
NETWORK
TITLE =
      AN    #Wejscie;
      L     S5T#5S;
      SD    #Timmer_2;
      NOP   0;
      NOP   0;
      NOP   0;
      NOP   0;
NETWORK
TITLE =
      A     #Wejscie;
      S     #Zmienna;
      A     #Wyjscie;
      R     #Zmienna;
      NOP   0;
END_FUNCTION

FUNCTION "Opoznienie_Wlotu" : VOID	// FC 86
VERSION : 0.1
VAR_INPUT
  Wejscie : BOOL ;	//Fotokomorka
  Timmer_1 : TIMER ;
  Timmer_2 : TIMER ;
END_VAR
VAR_OUTPUT
  Wyjscie : BOOL ;
END_VAR
VAR_IN_OUT
  Zmienna : BOOL ;
END_VAR
BEGIN
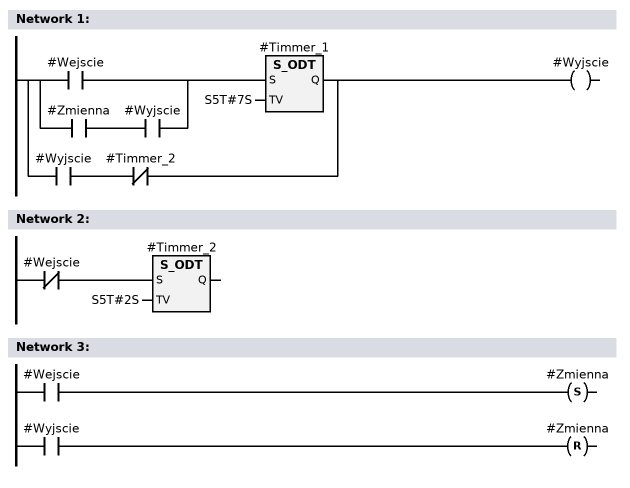
NETWORK
TITLE =
//Obecnosc palety jest aktywowana po 30s 
      O(;
      A(;
      O     #Wejscie;
      O;
      A     #Zmienna;
      A     #Wyjscie;
      );
      L     S5T#7S;
      SD    #Timmer_1;
      NOP   0;
      NOP   0;
      NOP   0;
      A     #Timmer_1;
      );
      O;
      A     #Wyjscie;
      AN    #Timmer_2;
      =     #Wyjscie;
NETWORK
TITLE =
//Filter 2s na fotokomorke aby nie zgasla gdy paleta jest na bandzie
      AN    #Wejscie;
      L     S5T#2S;
      SD    #Timmer_2;
      NOP   0;
      NOP   0;
      NOP   0;
      NOP   0;
NETWORK
TITLE =
      A     #Wejscie;
      S     #Zmienna;
      A     #Wyjscie;
      R     #Zmienna;
      NOP   0;
END_FUNCTION

FUNCTION "Komunikacja_GD" : VOID	// FC 100
VERSION : 0.1
BEGIN
NETWORK
TITLE =
//Ten network celowo jest wolny
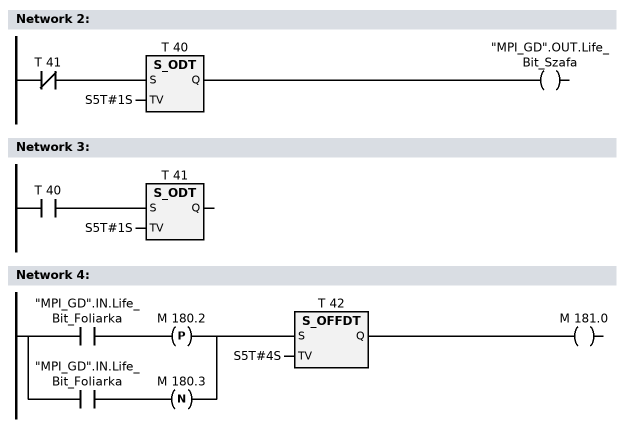
NETWORK
TITLE =
//Generator bit zycia foliarki
      AN    T 41;
      L     S5T#1S;
      SD    T 40;
      NOP   0;
      NOP   0;
      NOP   0;
      A     T 40;
      =     "MPI_GD".OUT.Life_Bit_Szafa;
NETWORK
TITLE =
//Generator bit zycia foliarki
      A     T 40;
      L     S5T#1S;
      SD    T 41;
      NOP   0;
      NOP   0;
      NOP   0;
      NOP   0;
NETWORK
TITLE =
//Sprawdzenie komunikacji z szafa transportera
      A(;
      A     "MPI_GD".IN.Life_Bit_Foliarka;
      FP    M 180.2;
      O(;
      A     "MPI_GD".IN.Life_Bit_Foliarka;
      FN    M 180.3;
      );
      );
      L     S5T#4S;
      SF    T 42;
      NOP   0;
      NOP   0;
      NOP   0;
      A     T 42;
      =     M 181.0;
END_FUNCTION

FUNCTION "Obsluga bledow" : VOID	// FC 119
VERSION : 0.1
BEGIN
NETWORK
TITLE =
//Ten network celowo jest wolny
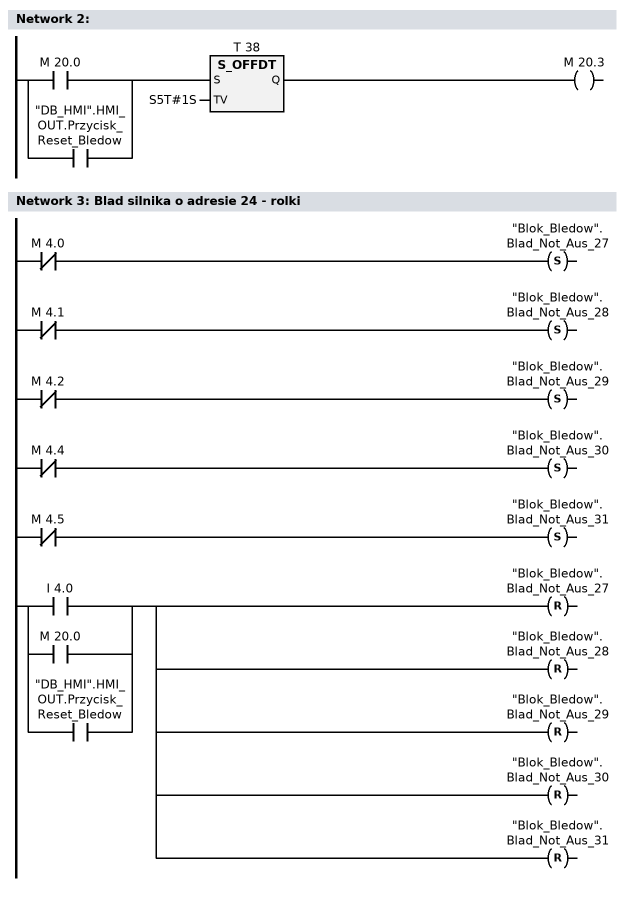
NETWORK
TITLE =
      A(;
      O     M 20.0;
      O     "DB_HMI".HMI_OUT.Przycisk_Reset_Bledow;
      );
      L     S5T#1S;
      SF    T 38;
      NOP   0;
      NOP   0;
      NOP   0;
      A     T 38;
      =     M 20.3;
NETWORK
TITLE = Blad silnika o adresie 24 - rolki
//Bledy do panelu HMI
//Not Aus 27*******************************
      AN    M 4.0;
      S     "Blok_Bledow".Blad_Not_Aus_27;
//Not Aus 28*******************************
      AN    M 4.1;
      S     "Blok_Bledow".Blad_Not_Aus_28;
//Not Aus 29*******************************
      AN    M 4.2;
      S     "Blok_Bledow".Blad_Not_Aus_29;
//Not Aus 30*******************************
      AN    M 4.4;
      S     "Blok_Bledow".Blad_Not_Aus_30;
//Not Aus 31*******************************
      AN    M 4.5;
      S     "Blok_Bledow".Blad_Not_Aus_31;
//Reset bledow not-aus
      O     I 4.0;
      O     M 20.0;
      O     "DB_HMI".HMI_OUT.Przycisk_Reset_Bledow;
      R     "Blok_Bledow".Blad_Not_Aus_27;
      R     "Blok_Bledow".Blad_Not_Aus_28;
      R     "Blok_Bledow".Blad_Not_Aus_29;
      R     "Blok_Bledow".Blad_Not_Aus_30;
      R     "Blok_Bledow".Blad_Not_Aus_31;
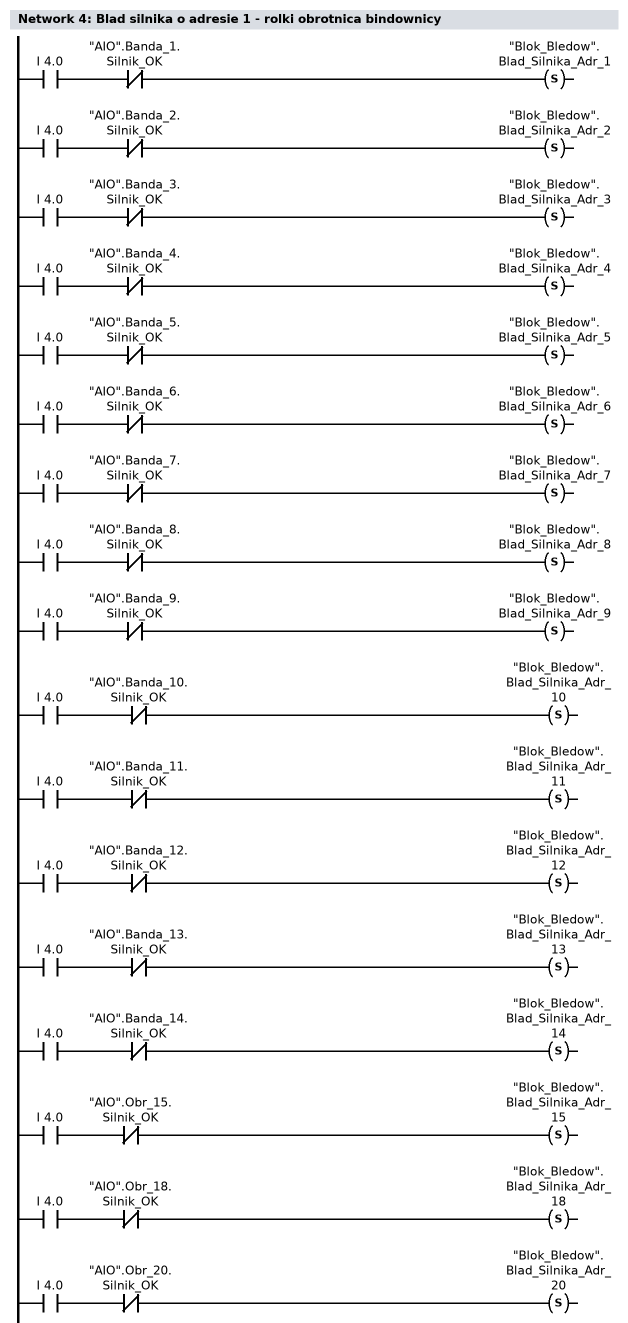
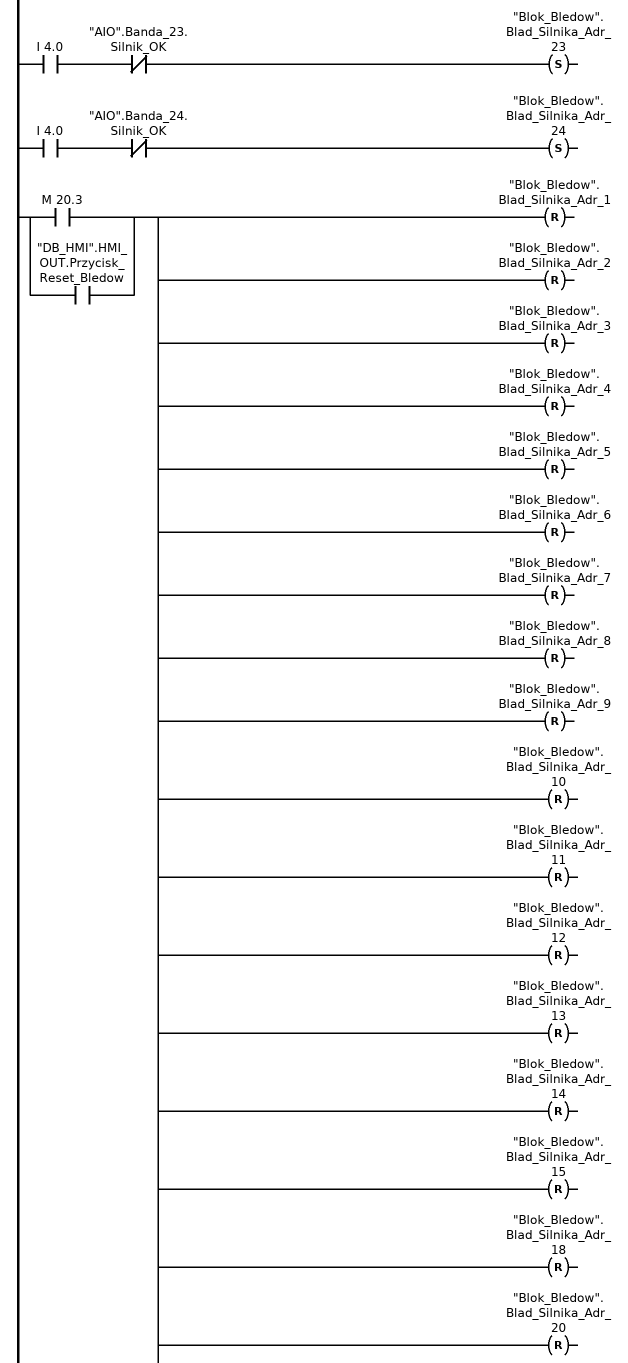
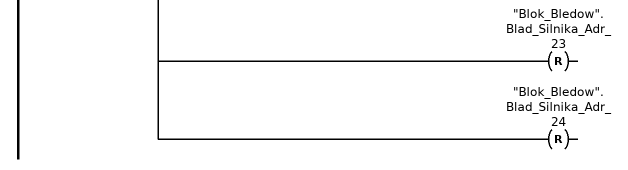
NETWORK
TITLE = Blad silnika o adresie 1 - rolki obrotnica bindownicy
//Bledy napedow
//Bledy napedow
      A     I 4.0;
      AN    "AIO".Banda_1.Silnik_OK;
      S     "Blok_Bledow".Blad_Silnika_Adr_1;
      A     I 4.0;
      AN    "AIO".Banda_2.Silnik_OK;
      S     "Blok_Bledow".Blad_Silnika_Adr_2;
      A     I 4.0;
      AN    "AIO".Banda_3.Silnik_OK;
      S     "Blok_Bledow".Blad_Silnika_Adr_3;
      A     I 4.0;
      AN    "AIO".Banda_4.Silnik_OK;
      S     "Blok_Bledow".Blad_Silnika_Adr_4;
      A     I 4.0;
      AN    "AIO".Banda_5.Silnik_OK;
      S     "Blok_Bledow".Blad_Silnika_Adr_5;
      A     I 4.0;
      AN    "AIO".Banda_6.Silnik_OK;
      S     "Blok_Bledow".Blad_Silnika_Adr_6;
      A     I 4.0;
      AN    "AIO".Banda_7.Silnik_OK;
      S     "Blok_Bledow".Blad_Silnika_Adr_7;
      A     I 4.0;
      AN    "AIO".Banda_8.Silnik_OK;
      S     "Blok_Bledow".Blad_Silnika_Adr_8;
      A     I 4.0;
      AN    "AIO".Banda_9.Silnik_OK;
      S     "Blok_Bledow".Blad_Silnika_Adr_9;
      A     I 4.0;
      AN    "AIO".Banda_10.Silnik_OK;
      S     "Blok_Bledow".Blad_Silnika_Adr_10;
      A     I 4.0;
      AN    "AIO".Banda_11.Silnik_OK;
      S     "Blok_Bledow".Blad_Silnika_Adr_11;
      A     I 4.0;
      AN    "AIO".Banda_12.Silnik_OK;
      S     "Blok_Bledow".Blad_Silnika_Adr_12;
      A     I 4.0;
      AN    "AIO".Banda_13.Silnik_OK;
      S     "Blok_Bledow".Blad_Silnika_Adr_13;
      A     I 4.0;
      AN    "AIO".Banda_14.Silnik_OK;
      S     "Blok_Bledow".Blad_Silnika_Adr_14;
      A     I 4.0;
      AN    "AIO".Obr_15.Silnik_OK;
      S     "Blok_Bledow".Blad_Silnika_Adr_15;
      A     I 4.0;
      AN    "AIO".Obr_18.Silnik_OK;
      S     "Blok_Bledow".Blad_Silnika_Adr_18;
      A     I 4.0;
      AN    "AIO".Obr_20.Silnik_OK;
      S     "Blok_Bledow".Blad_Silnika_Adr_20;
      A     I 4.0;
      AN    "AIO".Banda_23.Silnik_OK;
      S     "Blok_Bledow".Blad_Silnika_Adr_23;
      A     I 4.0;
      AN    "AIO".Banda_24.Silnik_OK;
      S     "Blok_Bledow".Blad_Silnika_Adr_24;
//Reset bledow napedow
//Reset bledow not-aus
      O     M 20.3;
      O     "DB_HMI".HMI_OUT.Przycisk_Reset_Bledow;
      R     "Blok_Bledow".Blad_Silnika_Adr_1;
      R     "Blok_Bledow".Blad_Silnika_Adr_2;
      R     "Blok_Bledow".Blad_Silnika_Adr_3;
      R     "Blok_Bledow".Blad_Silnika_Adr_4;
      R     "Blok_Bledow".Blad_Silnika_Adr_5;
      R     "Blok_Bledow".Blad_Silnika_Adr_6;
      R     "Blok_Bledow".Blad_Silnika_Adr_7;
      R     "Blok_Bledow".Blad_Silnika_Adr_8;
      R     "Blok_Bledow".Blad_Silnika_Adr_9;
      R     "Blok_Bledow".Blad_Silnika_Adr_10;
      R     "Blok_Bledow".Blad_Silnika_Adr_11;
      R     "Blok_Bledow".Blad_Silnika_Adr_12;
      R     "Blok_Bledow".Blad_Silnika_Adr_13;
      R     "Blok_Bledow".Blad_Silnika_Adr_14;
      R     "Blok_Bledow".Blad_Silnika_Adr_15;
      R     "Blok_Bledow".Blad_Silnika_Adr_18;
      R     "Blok_Bledow".Blad_Silnika_Adr_20;
      R     "Blok_Bledow".Blad_Silnika_Adr_23;
      R     "Blok_Bledow".Blad_Silnika_Adr_24;
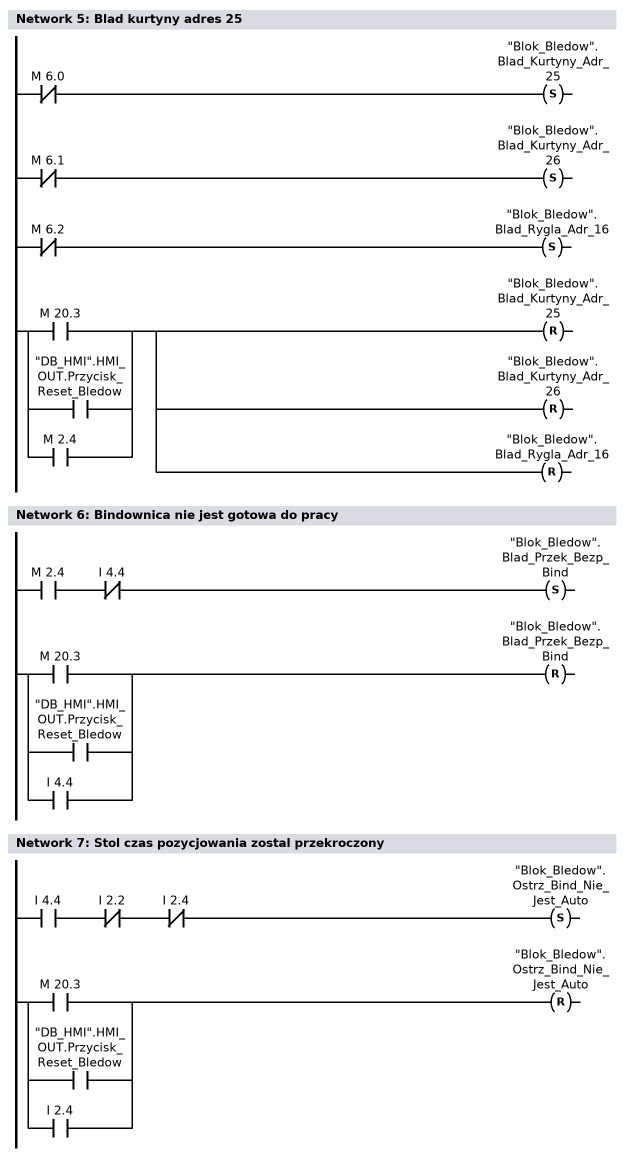
NETWORK
TITLE = Blad kurtyny adres 25
//Bledy kurtyn kasownie samoistne
      AN    M 6.0;
      S     "Blok_Bledow".Blad_Kurtyny_Adr_25;
      AN    M 6.1;
      S     "Blok_Bledow".Blad_Kurtyny_Adr_26;
      AN    M 6.2;
      S     "Blok_Bledow".Blad_Rygla_Adr_16;
      O     M 20.3;
      O     "DB_HMI".HMI_OUT.Przycisk_Reset_Bledow;
      O     M 2.4;
      R     "Blok_Bledow".Blad_Kurtyny_Adr_25;
      R     "Blok_Bledow".Blad_Kurtyny_Adr_26;
      R     "Blok_Bledow".Blad_Rygla_Adr_16;
NETWORK
TITLE = Bindownica nie jest gotowa do pracy
//Blad Przekaznika bezpieczenstwa kurtyn
      A     M 2.4;
      AN    I 4.4;
      S     "Blok_Bledow".Blad_Przek_Bezp_Bind;
      O     M 20.3;
      O     "DB_HMI".HMI_OUT.Przycisk_Reset_Bledow;
      O     I 4.4;
      R     "Blok_Bledow".Blad_Przek_Bezp_Bind;
NETWORK
TITLE = Stol czas pozycjowania zostal przekroczony
//Blad informacyjny bindownica nie jest w auto
      A     I 4.4;
      AN    I 2.2;
      AN    I 2.4;
      S     "Blok_Bledow".Ostrz_Bind_Nie_Jest_Auto;
      O     M 20.3;
      O     "DB_HMI".HMI_OUT.Przycisk_Reset_Bledow;
      O     I 2.4;
      R     "Blok_Bledow".Ostrz_Bind_Nie_Jest_Auto;
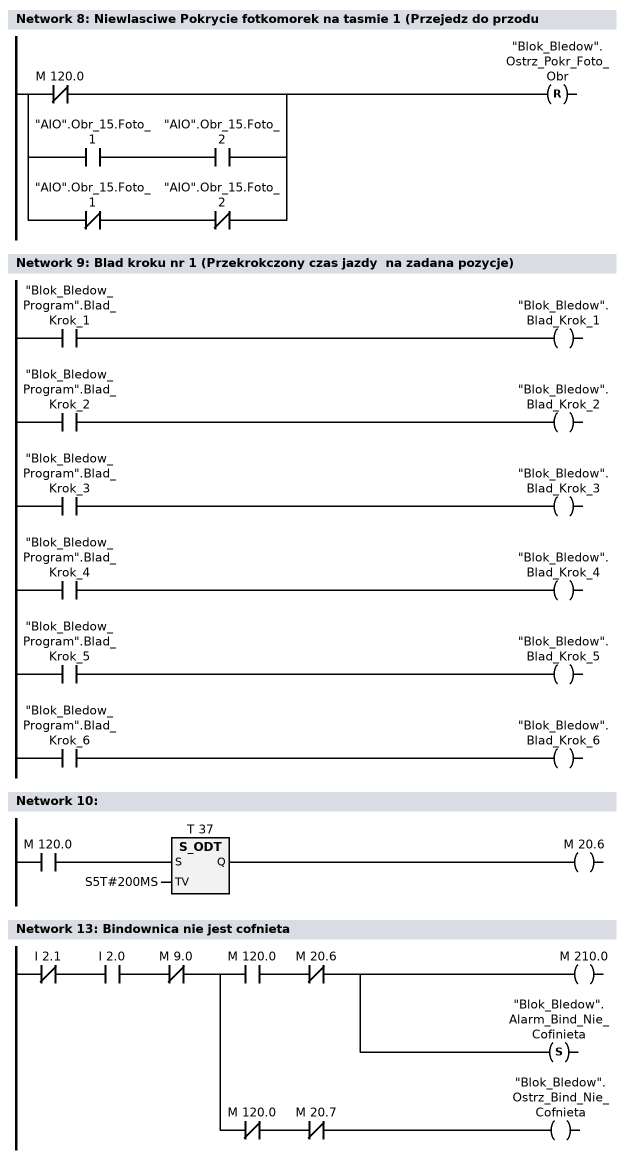
NETWORK
TITLE = Niewlasciwe Pokrycie fotkomorek na tasmie 1 (Przejedz do przodu 
//Ostrzezenie palety nie sa na fotokomorkach przednich
//
//Obrotnica
      ON    M 120.0;
      O;
      A     "AIO".Obr_15.Foto_1;
      A     "AIO".Obr_15.Foto_2;
      O;
      AN    "AIO".Obr_15.Foto_1;
      AN    "AIO".Obr_15.Foto_2;
      R     "Blok_Bledow".Ostrz_Pokr_Foto_Obr;
NETWORK
TITLE = Blad kroku nr 1 (Przekrokczony czas jazdy  na zadana pozycje)
//Bledy Zapalajaca czerwona lampke na panelu HMI
//Kwitowanie tych bledow przy pomocy przycisku. Reset nastepnie dalszy krok to 
//przywrocenie automatyki auto lub cyklem start
//
//
// Bledy czasu tranzycji krokow
      A     "Blok_Bledow_Program".Blad_Krok_1;
      =     "Blok_Bledow".Blad_Krok_1;
      A     "Blok_Bledow_Program".Blad_Krok_2;
      =     "Blok_Bledow".Blad_Krok_2;
      A     "Blok_Bledow_Program".Blad_Krok_3;
      =     "Blok_Bledow".Blad_Krok_3;
      A     "Blok_Bledow_Program".Blad_Krok_4;
      =     "Blok_Bledow".Blad_Krok_4;
      A     "Blok_Bledow_Program".Blad_Krok_5;
      =     "Blok_Bledow".Blad_Krok_5;
      A     "Blok_Bledow_Program".Blad_Krok_6;
      =     "Blok_Bledow".Blad_Krok_6;
NETWORK
TITLE =
//Wypadniecie maszyny z automatyki. Oraz powrot do polautomatu gdy automatyka nie 
//spelniona. 
      A     M 120.0;
      L     S5T#200MS;
      SD    T 37;
      NOP   0;
      NOP   0;
      NOP   0;
      A     T 37;
      =     M 20.6;
NETWORK
TITLE =
NETWORK
TITLE =
//Warunki sprawdzane podczas 200ms trybu Ghost Mode
//bity m210 w gore
NETWORK
TITLE = Bindownica nie jest cofnieta
//Bindownica nie jest w pozycji podstawoej
      AN    I 2.1;
      A     I 2.0;
      AN    M 9.0;
      =     L 0.0;
      A     L 0.0;
      A     M 120.0;
      AN    M 20.6;
      =     M 210.0;
      S     "Blok_Bledow".Alarm_Bind_Nie_Cofinieta;
      A     L 0.0;
      AN    M 120.0;
      AN    M 20.7;
      =     "Blok_Bledow".Ostrz_Bind_Nie_Cofnieta;
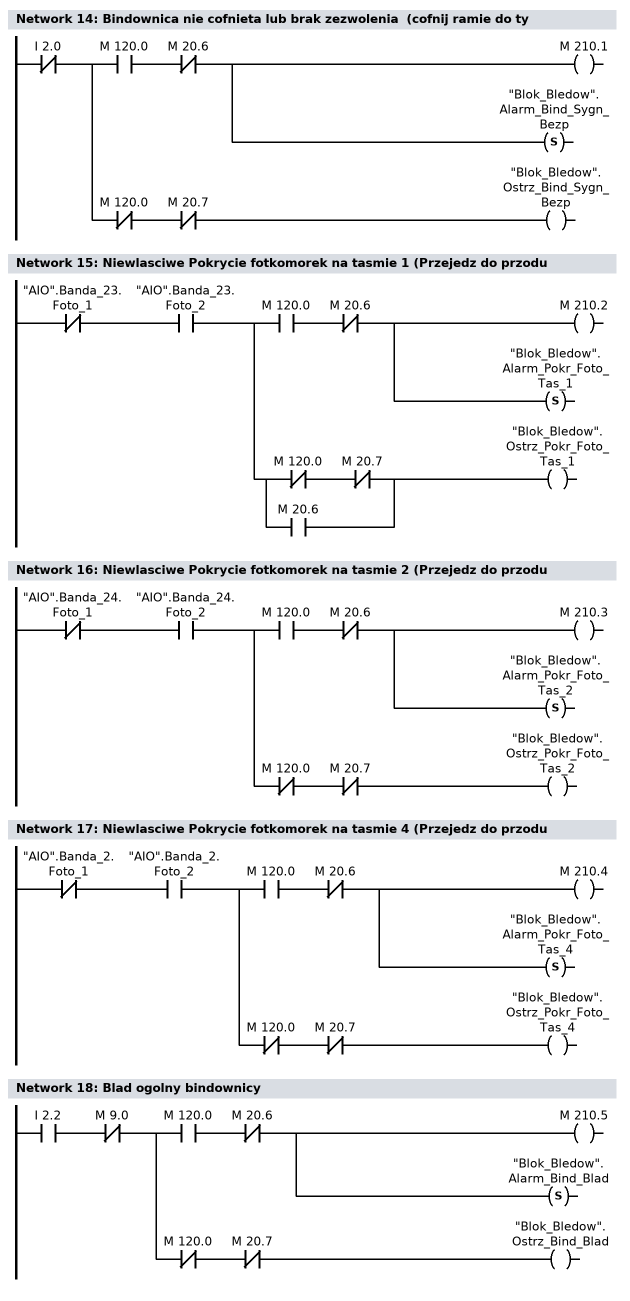
NETWORK
TITLE = Bindownica nie cofnieta lub brak zezwolenia  (cofnij ramie do ty
//Bindownica nie daje sygnalu bezpieczestwa
      AN    I 2.0;
      =     L 0.0;
      A     L 0.0;
      A     M 120.0;
      AN    M 20.6;
      =     M 210.1;
      S     "Blok_Bledow".Alarm_Bind_Sygn_Bezp;
      A     L 0.0;
      AN    M 120.0;
      AN    M 20.7;
      =     "Blok_Bledow".Ostrz_Bind_Sygn_Bezp;
NETWORK
TITLE = Niewlasciwe Pokrycie fotkomorek na tasmie 1 (Przejedz do przodu 
//Tasma 1 Wyjatek bo tutaj kladzie sie palete w automacie przez wozek
      AN    "AIO".Banda_23.Foto_1;
      A     "AIO".Banda_23.Foto_2;
      =     L 0.0;
      A     L 0.0;
      A     M 120.0;
      AN    M 20.6;
      =     M 210.2;
      S     "Blok_Bledow".Alarm_Pokr_Foto_Tas_1;
      A     L 0.0;
      A(;
      AN    M 120.0;
      AN    M 20.7;
      O     M 20.6;
      );
      =     "Blok_Bledow".Ostrz_Pokr_Foto_Tas_1;
NETWORK
TITLE = Niewlasciwe Pokrycie fotkomorek na tasmie 2 (Przejedz do przodu 
//Tasma 2   O     "DB_HMI".HMI_OUT.Przycisk_Reset_Bledow
      AN    "AIO".Banda_24.Foto_1;
      A     "AIO".Banda_24.Foto_2;
      =     L 0.0;
      A     L 0.0;
      A     M 120.0;
      AN    M 20.6;
      =     M 210.3;
      S     "Blok_Bledow".Alarm_Pokr_Foto_Tas_2;
      A     L 0.0;
      AN    M 120.0;
      AN    M 20.7;
      =     "Blok_Bledow".Ostrz_Pokr_Foto_Tas_2;
NETWORK
TITLE = Niewlasciwe Pokrycie fotkomorek na tasmie 4 (Przejedz do przodu 
//Tasma:4      "DB_HMI".HMI_OUT.Przycisk_Reset_Bledow
      AN    "AIO".Banda_2.Foto_1;
      A     "AIO".Banda_2.Foto_2;
      =     L 0.0;
      A     L 0.0;
      A     M 120.0;
      AN    M 20.6;
      =     M 210.4;
      S     "Blok_Bledow".Alarm_Pokr_Foto_Tas_4;
      A     L 0.0;
      AN    M 120.0;
      AN    M 20.7;
      =     "Blok_Bledow".Ostrz_Pokr_Foto_Tas_4;
NETWORK
TITLE = Blad ogolny bindownicy 
//Blad ogolny bindownicy
      A     I 2.2;
      AN    M 9.0;
      =     L 0.0;
      A     L 0.0;
      A     M 120.0;
      AN    M 20.6;
      =     M 210.5;
      S     "Blok_Bledow".Alarm_Bind_Blad;
      A     L 0.0;
      AN    M 120.0;
      AN    M 20.7;
      =     "Blok_Bledow".Ostrz_Bind_Blad;
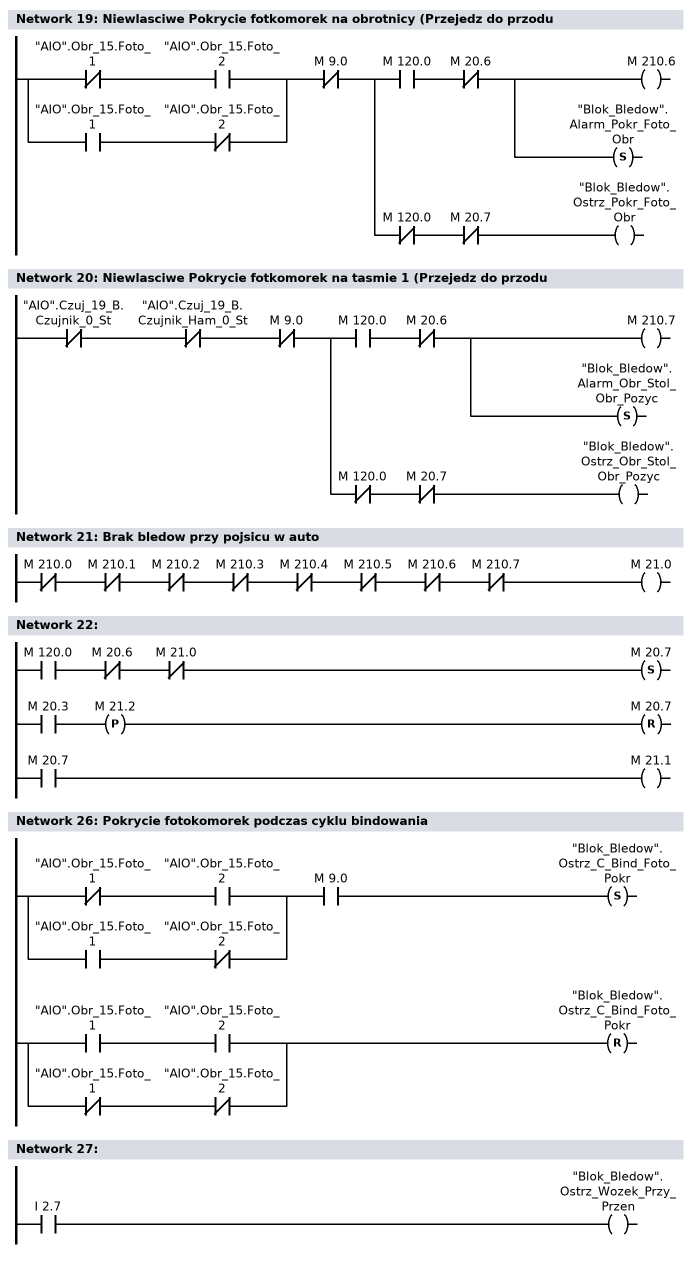
NETWORK
TITLE = Niewlasciwe Pokrycie fotkomorek na obrotnicy (Przejedz do przodu
//Blad fotokomorek stolu obrotowego
      A(;
      AN    "AIO".Obr_15.Foto_1;
      A     "AIO".Obr_15.Foto_2;
      O;
      A     "AIO".Obr_15.Foto_1;
      AN    "AIO".Obr_15.Foto_2;
      );
      AN    M 9.0;
      =     L 0.0;
      A     L 0.0;
      A     M 120.0;
      AN    M 20.6;
      =     M 210.6;
      S     "Blok_Bledow".Alarm_Pokr_Foto_Obr;
      A     L 0.0;
      AN    M 120.0;
      AN    M 20.7;
      =     "Blok_Bledow".Ostrz_Pokr_Foto_Obr;
NETWORK
TITLE = Niewlasciwe Pokrycie fotkomorek na tasmie 1 (Przejedz do przodu 
//Stol obrotowy nie w pozycji
      AN    "AIO".Czuj_19_B.Czujnik_0_St;
      AN    "AIO".Czuj_19_B.Czujnik_Ham_0_St;
      AN    M 9.0;
      =     L 0.0;
      A     L 0.0;
      A     M 120.0;
      AN    M 20.6;
      =     M 210.7;
      S     "Blok_Bledow".Alarm_Obr_Stol_Obr_Pozyc;
      A     L 0.0;
      AN    M 120.0;
      AN    M 20.7;
      =     "Blok_Bledow".Ostrz_Obr_Stol_Obr_Pozyc;
NETWORK
TITLE = Brak bledow przy pojsicu w auto
//Sprawdzam
      AN    M 210.0;
      AN    M 210.1;
      AN    M 210.2;
      AN    M 210.3;
      AN    M 210.4;
      AN    M 210.5;
      AN    M 210.6;
      AN    M 210.7;
      =     M 21.0;
NETWORK
TITLE =
//Powrot do stopu polautomatu jesli jest blad
      A     M 120.0;
      AN    M 20.6;
      AN    M 21.0;
      S     M 20.7;
      A     M 20.3;
      FP    M 21.2;
      R     M 20.7;
      A     M 20.7;
      =     M 21.1;
NETWORK
TITLE = Bindownica nie cofnieta lub brak zezwolenia  (cofnij ramie do ty
//reset komunikatow
//
      A     M 20.3;
//Alarmy
      R     "Blok_Bledow".Alarm_Obr_Stol_Obr_Pozyc;
      R     "Blok_Bledow".Alarm_Bind_Nie_Cofinieta;
      R     "Blok_Bledow".Alarm_Bind_Sygn_Bezp;
      R     "Blok_Bledow".rez3;
      R     "Blok_Bledow".rez_6_0;
      R     "Blok_Bledow".Alarm_Pokr_Foto_Tas_1;
      R     "Blok_Bledow".Alarm_Pokr_Foto_Tas_2;
      R     "Blok_Bledow".Alarm_Pokr_Foto_Tas_4;
      R     "Blok_Bledow".Alarm_Pokr_Foto_Obr;
      R     "Blok_Bledow".Alarm_Bind_Nie_Jest_Auto;
      R     "Blok_Bledow".Alarm_Bind_Blad;
      R     "Blok_Bledow".rez_6_7;
      R     "Blok_Bledow".Ostrz_Prasa_Nie_W_Gorze;
      R     "Blok_Bledow".rez_7_1;
//Warnings
      R     "Blok_Bledow".Ostrz_Bind_Blad;
      R     "Blok_Bledow".Ostrz_Bind_Nie_Cofnieta;
      R     "Blok_Bledow".Ostrz_Bind_Sygn_Bezp;
      R     "Blok_Bledow".Ostrz_Bind_Nie_Jest_Auto;
      R     "Blok_Bledow".Ostrz_Stol_Obr_Foto;
      R     "Blok_Bledow".Ostrz_Obr_Stol_Obr_Pozyc;
      R     "Blok_Bledow".Ostrz_Pokr_Foto_Tas_1;
      R     "Blok_Bledow".Ostrz_Pokr_Foto_Tas_2;
      R     "Blok_Bledow".Ostrz_Pokr_Foto_Obr;
      R     "Blok_Bledow".Ostrz_Pokr_Foto_Tas_4;
      CLR;
NETWORK
TITLE =
//Koniec sprawdzanie wejscia w automatyke
NETWORK
TITLE =
//Sprawdzenie maszyny podczas cyklu. Zwracane sa ostrzezenia by byla informacja 
//ale nie przerwac dzialania
NETWORK
TITLE = Pokrycie fotokomorek podczas cyklu bindowania
//Niewlasciwe pokrycie fotokomorek podczas cyklu
      A(;
      AN    "AIO".Obr_15.Foto_1;
      A     "AIO".Obr_15.Foto_2;
      O;
      A     "AIO".Obr_15.Foto_1;
      AN    "AIO".Obr_15.Foto_2;
      );
      A     M 9.0;
      S     "Blok_Bledow".Ostrz_C_Bind_Foto_Pokr;
      A(;
      A     "AIO".Obr_15.Foto_1;
      A     "AIO".Obr_15.Foto_2;
      O;
      AN    "AIO".Obr_15.Foto_1;
      AN    "AIO".Obr_15.Foto_2;
      );
      R     "Blok_Bledow".Ostrz_C_Bind_Foto_Pokr;
      NOP   0;
NETWORK
TITLE =
//Cykl trwa a bindownica nie jest z tylu
      A     I 2.7;
      =     "Blok_Bledow".Ostrz_Wozek_Przy_Przen;
